REGION Network 2: Инициализация
   // При первом включении проверка наличия аварий и перегрева.
   // При перегреве --  охлаждение. Если долго не остывает, то авария.
   RUNG wire#powerrail
      "Initializing&Cooling_DB"(resetTrigg := wire#w1, iniOk => "Main_PRG".iniOk, initializing => "Main_PRG".initializing, faultTrigg => "READ".status.errorTrigg, warning => "READ".status.warning, toAirClean => #iniAir, toCoolUpLaser => #iniUpLaser, toCoolUpCam => #iniUpCam, toCoolDownLaser => #iniDownLaser, toCoolDownCam => #iniDownCam)
   END_RUNG
   RUNG wire#powerrail
      Contact( "WRITE".resetErrorTrigg )
   END_RUNG wire#w1
   RUNG wire#powerrail
      Contact( "READ".inputs.resetAlm )
   END_RUNG wire#w1
   // the same network as SCL:
   "Initializing&Cooling_DB"(resetTrigg := "WRITE".resetErrorTrigg OR "READ".inputs.resetAlm,   // "Initializing&Cooling"
                           iniOk => "Main_PRG".iniOk,
                           initializing => "Main_PRG".initializing,
                           faultTrigg => "READ".status.errorTrigg,
                           warning => "READ".status.warning,
                           toAirClean => #iniAir,
                           toCoolUpLaser => #iniUpLaser,
                           toCoolUpCam => #iniUpCam,
                           toCoolDownLaser => #iniDownLaser,
                           toCoolDownCam => #iniDownCam);
END_REGION

REGION Network 3: Основная программа
   // Включение велосиметра, обдува, охлаждения, сигналов ламп
   RUNG wire#powerrail
      "Main_Block_db"(faultTrigg := "READ".status.errorTrigg, warning := "READ".status.warning, initializing := "Main_PRG".initializing, initOk := "Main_PRG".iniOk, outEnable := "READ".inputs.runForward, velocimeterModeManual := "READ".inputs.veloModeManual, velocimeterModeAuto := "READ".inputs.veloModeAuto, revers := "READ".inputs.runBackward, synchroOn := "Main_PRG".synchroOn, airTon := "WRITE".cleanTime.tOnS, airToff := "WRITE".cleanTime.tOffMin, speed := "READ".velometer.instSpeed, RUN => "Main_PRG".RUN, airOn => #autoAir, veloLaser_En => "READ".outputs.disVelocimeter, veloShut_En => "READ".outputs.enVelocimeter, coolUpLaserOn => #autoUpLaser, coolUpCamOn => #autoUpCam, coolDownLaserOn => #autoDownLaser, coolDownCamOn => #autoDownCam, redLamp => "READ".outputs.redLamp, greenLamp => "READ".outputs.greenLamp, dirForward => "READ".status.veloPositive, dirBackward => "READ".status.veloNegative, greenLampStat => "READ".status.greenLamp, redLampStat => "READ".status.redLamp)
   END_RUNG
   // the same network as SCL:
   "Main_Block_db"(faultTrigg := "READ".status.errorTrigg,   // "Main_Block"
                   warning := "READ".status.warning,
                   initializing := "Main_PRG".initializing,
                   initOk := "Main_PRG".iniOk,
                   outEnable := "READ".inputs.runForward,
                   velocimeterModeManual := "READ".inputs.veloModeManual,
                   velocimeterModeAuto := "READ".inputs.veloModeAuto,
                   revers := "READ".inputs.runBackward,
                   synchroOn := "Main_PRG".synchroOn,
                   airTon := "WRITE".cleanTime.tOnS,
                   airToff := "WRITE".cleanTime.tOffMin,
                   speed := "READ".velometer.instSpeed,
                   RUN => "Main_PRG".RUN,
                   airOn => #autoAir,
                   veloLaser_En => "READ".outputs.disVelocimeter,
                   veloShut_En => "READ".outputs.enVelocimeter,
                   coolUpLaserOn => #autoUpLaser,
                   coolUpCamOn => #autoUpCam,
                   coolDownLaserOn => #autoDownLaser,
                   coolDownCamOn => #autoDownCam,
                   redLamp => "READ".outputs.redLamp,
                   greenLamp => "READ".outputs.greenLamp,
                   dirForward => "READ".status.veloPositive,
                   dirBackward => "READ".status.veloNegative,
                   greenLampStat => "READ".status.greenLamp,
                   redLampStat => "READ".status.redLamp);
END_REGION

REGION Network 4: Включение лазеров и синхронизации
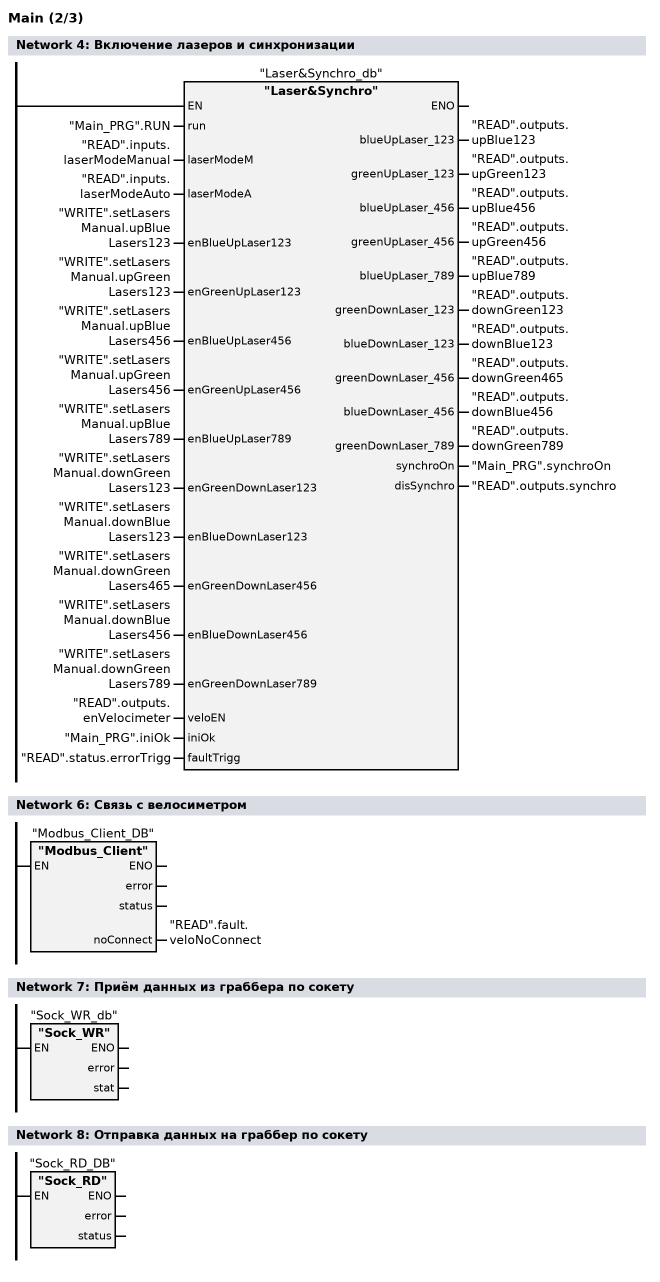
   RUNG wire#powerrail
      "Laser&Synchro_db"(run := "Main_PRG".RUN, laserModeM := "READ".inputs.laserModeManual, laserModeA := "READ".inputs.laserModeAuto, enBlueUpLaser123 := "WRITE".setLasersManual.upBlueLasers123, enGreenUpLaser123 := "WRITE".setLasersManual.upGreenLasers123, enBlueUpLaser456 := "WRITE".setLasersManual.upBlueLasers456, enGreenUpLaser456 := "WRITE".setLasersManual.upGreenLasers456, enBlueUpLaser789 := "WRITE".setLasersManual.upBlueLasers789, enGreenDownLaser123 := "WRITE".setLasersManual.downGreenLasers123, enBlueDownLaser123 := "WRITE".setLasersManual.downBlueLasers123, enGreenDownLaser456 := "WRITE".setLasersManual.downGreenLasers465, enBlueDownLaser456 := "WRITE".setLasersManual.downBlueLasers456, enGreenDownLaser789 := "WRITE".setLasersManual.downGreenLasers789, veloEN := "READ".outputs.enVelocimeter, iniOk := "Main_PRG".iniOk, faultTrigg := "READ".status.errorTrigg, blueUpLaser_123 => "READ".outputs.upBlue123, greenUpLaser_123 => "READ".outputs.upGreen123, blueUpLaser_456 => "READ".outputs.upBlue456, greenUpLaser_456 => "READ".outputs.upGreen456, blueUpLaser_789 => "READ".outputs.upBlue789, greenDownLaser_123 => "READ".outputs.downGreen123, blueDownLaser_123 => "READ".outputs.downBlue123, greenDownLaser_456 => "READ".outputs.downGreen465, blueDownLaser_456 => "READ".outputs.downBlue456, greenDownLaser_789 => "READ".outputs.downGreen789, synchroOn => "Main_PRG".synchroOn, disSynchro => "READ".outputs.synchro)
   END_RUNG
   // the same network as SCL:
   "Laser&Synchro_db"(run := "Main_PRG".RUN,   // "Laser&Synchro"
                      laserModeM := "READ".inputs.laserModeManual,
                      laserModeA := "READ".inputs.laserModeAuto,
                      enBlueUpLaser123 := "WRITE".setLasersManual.upBlueLasers123,
                      enGreenUpLaser123 := "WRITE".setLasersManual.upGreenLasers123,
                      enBlueUpLaser456 := "WRITE".setLasersManual.upBlueLasers456,
                      enGreenUpLaser456 := "WRITE".setLasersManual.upGreenLasers456,
                      enBlueUpLaser789 := "WRITE".setLasersManual.upBlueLasers789,
                      enGreenDownLaser123 := "WRITE".setLasersManual.downGreenLasers123,
                      enBlueDownLaser123 := "WRITE".setLasersManual.downBlueLasers123,
                      enGreenDownLaser456 := "WRITE".setLasersManual.downGreenLasers465,
                      enBlueDownLaser456 := "WRITE".setLasersManual.downBlueLasers456,
                      enGreenDownLaser789 := "WRITE".setLasersManual.downGreenLasers789,
                      veloEN := "READ".outputs.enVelocimeter,
                      iniOk := "Main_PRG".iniOk,
                      faultTrigg := "READ".status.errorTrigg,
                      blueUpLaser_123 => "READ".outputs.upBlue123,
                      greenUpLaser_123 => "READ".outputs.upGreen123,
                      blueUpLaser_456 => "READ".outputs.upBlue456,
                      greenUpLaser_456 => "READ".outputs.upGreen456,
                      blueUpLaser_789 => "READ".outputs.upBlue789,
                      greenDownLaser_123 => "READ".outputs.downGreen123,
                      blueDownLaser_123 => "READ".outputs.downBlue123,
                      greenDownLaser_456 => "READ".outputs.downGreen465,
                      blueDownLaser_456 => "READ".outputs.downBlue456,
                      greenDownLaser_789 => "READ".outputs.downGreen789,
                      synchroOn => "Main_PRG".synchroOn,
                      disSynchro => "READ".outputs.synchro);
END_REGION

REGION Network 5 (SCL): Объединение сигналов
   "READ".outputs.airClean := #iniAir OR #autoAir;
   "READ".outputs.coolUpLaser := #iniUpLaser OR #autoUpLaser;
   "READ".outputs.coolUpCam := #iniUpCam OR #autoUpCam;
   "READ".outputs.coolDownLaser := #iniDownLaser OR #autoDownLaser;
   "READ".outputs.coolDownCam := #iniDownCam OR #autoDownCam;
END_REGION

REGION Network 6: Связь с велосиметром
   RUNG wire#powerrail
      "Modbus_Client_DB"(error =>, status =>, noConnect => "READ".fault.veloNoConnect)
   END_RUNG
   // the same network as SCL:
   "Modbus_Client_DB"(noConnect => "READ".fault.veloNoConnect);   // "Modbus_Client"
END_REGION

REGION Network 7: Приём данных из граббера по сокету
   RUNG wire#powerrail
      "Sock_WR_db"(error =>, stat =>)
   END_RUNG
   // the same network as SCL:
   "Sock_WR_db"();   // "Sock_WR"
END_REGION

REGION Network 8: Отправка данных на граббер по сокету
   RUNG wire#powerrail
      "Sock_RD_DB"(error =>, status =>)
   END_RUNG
   // the same network as SCL:
   "Sock_RD_DB"();   // "Sock_RD"
END_REGION

REGION Network 9: Включение охладителя воздуха пневмосистемы
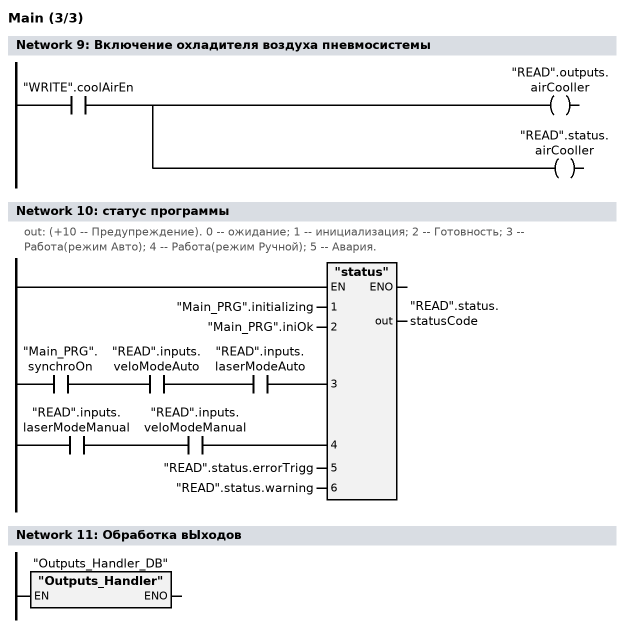
   RUNG wire#powerrail
      Contact( "WRITE".coolAirEn )
      wire#w1
      Coil( "READ".outputs.airCooller )
   END_RUNG
   RUNG wire#w1
      Coil( "READ".status.airCooller )
   END_RUNG
   // the same network as SCL:
   "READ".outputs.airCooller := "WRITE".coolAirEn;
   "READ".status.airCooller := "WRITE".coolAirEn;
END_REGION

REGION Network 10: статус программы
   // out: (+10 -- Предупреждение). 0 -- ожидание; 1 -- инициализация; 2 -- Готовность; 3 -- Работа(режим Авто); 4 -- Работа(режим Ручной); 5 -- Авария.
   RUNG wire#powerrail
      "status"("3" := wire#w1, "4" := wire#w2, "1" := "Main_PRG".initializing, "2" := "Main_PRG".iniOk, "5" := "READ".status.errorTrigg, "6" := "READ".status.warning, out => "READ".status.statusCode)
   END_RUNG
   RUNG wire#powerrail
      Contact( "Main_PRG".synchroOn )
      Contact( "READ".inputs.veloModeAuto )
      Contact( "READ".inputs.laserModeAuto )
   END_RUNG wire#w1
   RUNG wire#powerrail
      Contact( "READ".inputs.laserModeManual )
      Contact( "READ".inputs.veloModeManual )
   END_RUNG wire#w2
   // the same network as SCL:
   "status"("1" := "Main_PRG".initializing,
            "2" := "Main_PRG".iniOk,
            "3" := "Main_PRG".synchroOn AND "READ".inputs.veloModeAuto AND "READ".inputs.laserModeAuto,
            "4" := "READ".inputs.laserModeManual AND "READ".inputs.veloModeManual,
            "5" := "READ".status.errorTrigg,
            "6" := "READ".status.warning,
            out => "READ".status.statusCode);
END_REGION

REGION Network 11: Обработка вЫходов
   RUNG wire#powerrail
      "Outputs_Handler_DB"()
   END_RUNG
   // the same network as SCL:
   "Outputs_Handler_DB"();   // "Outputs_Handler"
END_REGION
END_ORGANIZATION_BLOCK

// folder: FBlocks

FUNCTION_BLOCK "Decode8toBool"   // FB2, SCL
{ S7_Optimized_Access := 'TRUE' }
VERSION : 0.1
   VAR_INPUT
      in : Byte;
   END_VAR
   VAR_OUTPUT
      b0 : Bool;
      b1 : Bool;
      b2 : Bool;
      b3 : Bool;
      b4 : Bool;
      b5 : Bool;
      b6 : Bool;
      b7 : Bool;
      "OR" : Bool;
   END_VAR
   VAR
      boolArray : Array[0..7] of Bool;
      i : USInt;
      "m" : USInt;
      temp : UDInt;
   END_VAR
BEGIN
   FOR #i := 0 TO 7 DO
       "MOD"(in0 := #in,
             in1 := 2,
             Out => #m);
       IF #m > 0 THEN
           #boolArray[#i] := TRUE;
       ELSE
           #boolArray[#i] := FALSE;
       END_IF;
       #in := #in / 2;
   END_FOR;

   #b0 := #boolArray[0];
   #b1 := #boolArray[1];
   #b2 := #boolArray[2];
   #b3 := #boolArray[3];
   #b4 := #boolArray[4];
   #b5 := #boolArray[5];
   #b6 := #boolArray[6];
   #b7 := #boolArray[7];

   #OR := #b2 OR #b4 OR #b6 OR #b7;
END_FUNCTION_BLOCK

FUNCTION_BLOCK "Hysteresis"   // FB4, LAD
{ S7_Optimized_Access := 'TRUE' }
VERSION : 0.1
   VAR_INPUT
      in : Real;
      SP : Real;
      hyster : Real;
   END_VAR
   VAR_OUTPUT
      cold : Bool;
      warm : Bool;
   END_VAR
   VAR_TEMP
      upperThreshold : Real;
      lowerThreshold : Real;
   END_VAR
BEGIN

REGION Network 1 (SCL)
   #upperThreshold := #SP + (#hyster / 2);
   #lowerThreshold := #SP - (#hyster / 2);

   IF #in > #upperThreshold THEN
       #cold := true;
       #warm := false;
   ELSIF #in < #lowerThreshold THEN
       #cold := false;
       #warm := true;
   END_IF;
END_REGION
END_FUNCTION_BLOCK

FUNCTION_BLOCK "4Hysteresis"   // FB5, LAD
{ S7_Optimized_Access := 'TRUE' }
VERSION : 0.1
   VAR_INPUT
      in0 : Real;
      in1 : Real := 0.0;
      in2 : Real := 0.0;
      in3 : Real := 0.0;
      SP0 : Real;
      SP1 : Real := 0.0;
      SP2 : Real := 0.0;
      SP3 : Real := 0.0;
      hyster : Real;
      TON : Time;
   END_VAR
   VAR_OUTPUT
      out0 : Bool;
      out1 : Bool := false;
      out2 : Bool := false;
      out3 : Bool := false;
   END_VAR
   VAR
      Hysteresis_Instance : "Hysteresis";
      Hysteresis_Instance_1 : "Hysteresis";
      Hysteresis_Instance_2 : "Hysteresis";
      Hysteresis_Instance_3 : "Hysteresis";
      IEC_Timer_0_Instance : TON_TIME;
      IEC_Timer_0_Instance_1 : TON_TIME;
      IEC_Timer_0_Instance_2 : TON_TIME;
      IEC_Timer_0_Instance_3 : TON_TIME;
   END_VAR
   VAR_TEMP
      gi0 : Bool;
      gi1 : Bool;
      gi2 : Bool;
      gi3 : Bool;
   END_VAR
BEGIN

REGION Network 1
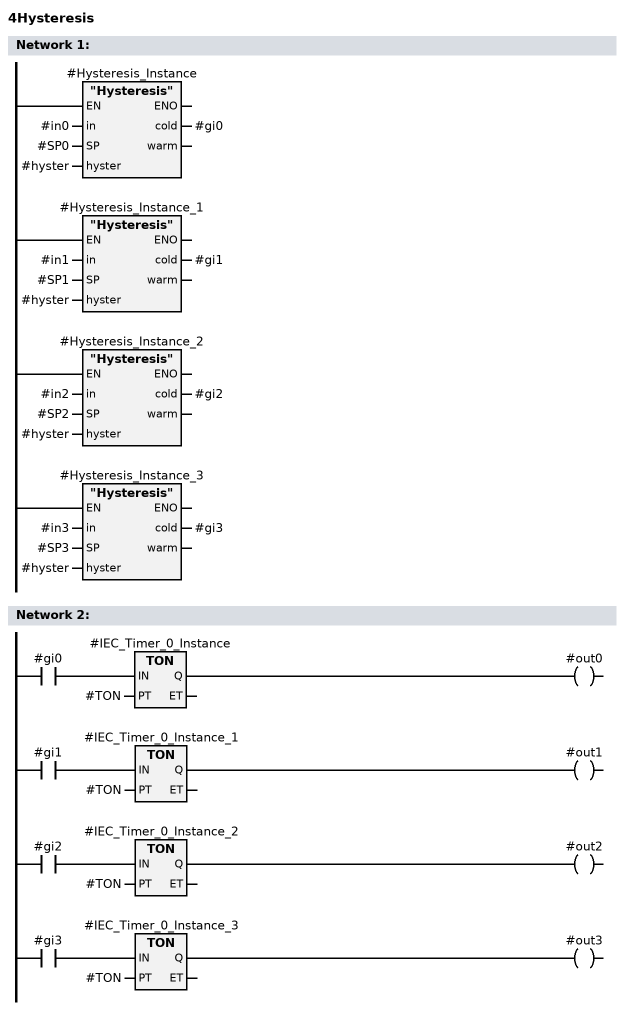
   RUNG wire#powerrail
      #Hysteresis_Instance(in := #in0, SP := #SP0, hyster := #hyster, cold => #gi0, warm =>)
   END_RUNG
   RUNG wire#powerrail
      #Hysteresis_Instance_1(in := #in1, SP := #SP1, hyster := #hyster, cold => #gi1, warm =>)
   END_RUNG
   RUNG wire#powerrail
      #Hysteresis_Instance_2(in := #in2, SP := #SP2, hyster := #hyster, cold => #gi2, warm =>)
   END_RUNG
   RUNG wire#powerrail
      #Hysteresis_Instance_3(in := #in3, SP := #SP3, hyster := #hyster, cold => #gi3, warm =>)
   END_RUNG
   // the same network as SCL:
   #Hysteresis_Instance(in := #in0, SP := #SP0, hyster := #hyster, cold => #gi0);   // "Hysteresis"
   #Hysteresis_Instance_1(in := #in1, SP := #SP1, hyster := #hyster, cold => #gi1);   // "Hysteresis"
   #Hysteresis_Instance_2(in := #in2, SP := #SP2, hyster := #hyster, cold => #gi2);   // "Hysteresis"
   #Hysteresis_Instance_3(in := #in3, SP := #SP3, hyster := #hyster, cold => #gi3);   // "Hysteresis"
END_REGION

REGION Network 2
   #IEC_Timer_0_Instance(IN := #gi0, PT := #TON);   // TON
   #out0 := #IEC_Timer_0_Instance.Q;
   #IEC_Timer_0_Instance_1(IN := #gi1, PT := #TON);   // TON
   #out1 := #IEC_Timer_0_Instance_1.Q;
   #IEC_Timer_0_Instance_2(IN := #gi2, PT := #TON);   // TON
   #out2 := #IEC_Timer_0_Instance_2.Q;
   #IEC_Timer_0_Instance_3(IN := #gi3, PT := #TON);   // TON
   #out3 := #IEC_Timer_0_Instance_3.Q;
END_REGION
END_FUNCTION_BLOCK

FUNCTION_BLOCK "5Hysteresis"   // FB6, LAD
{ S7_Optimized_Access := 'TRUE' }
VERSION : 0.1
   VAR_INPUT
      in0 : Real;
      in1 : Real := 0.0;
      in2 : Real := 0.0;
      in3 : Real := 0.0;
      in4 : Real := 0.0;
      SP0 : Real;
      SP1 : Real := 0.0;
      SP2 : Real := 0.0;
      SP3 : Real := 0.0;
      SP4 : Real := 0.0;
      hyster : Real;
   END_VAR
   VAR_OUTPUT
      out0 : Bool;
      out1 : Bool := false;
      out2 : Bool := false;
      out3 : Bool := false;
      out4 : Bool := false;
   END_VAR
   VAR
      Hysteresis_Instance : "Hysteresis";
      Hysteresis_Instance_1 : "Hysteresis";
      Hysteresis_Instance_2 : "Hysteresis";
      Hysteresis_Instance_3 : "Hysteresis";
      Hysteresis_Instance_4 : "Hysteresis";
   END_VAR
BEGIN

REGION Network 1
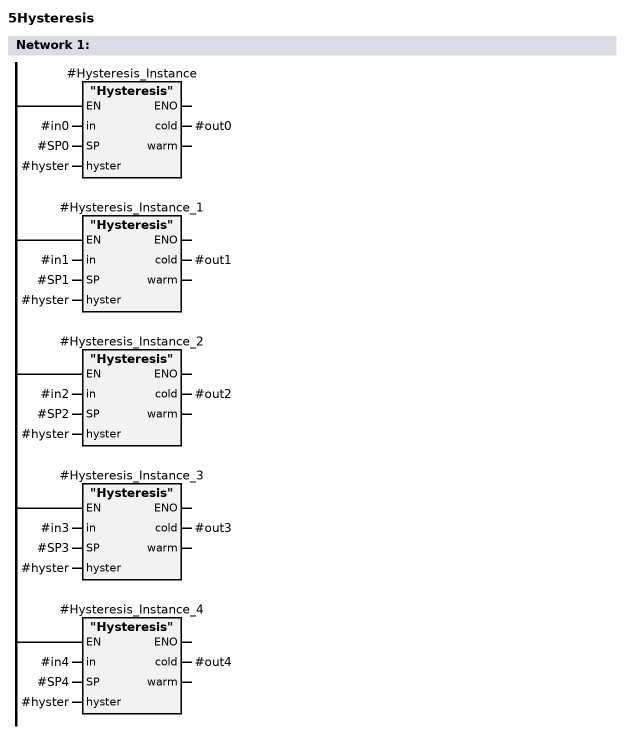
   RUNG wire#powerrail
      #Hysteresis_Instance(in := #in0, SP := #SP0, hyster := #hyster, cold => #out0, warm =>)
   END_RUNG
   RUNG wire#powerrail
      #Hysteresis_Instance_1(in := #in1, SP := #SP1, hyster := #hyster, cold => #out1, warm =>)
   END_RUNG
   RUNG wire#powerrail
      #Hysteresis_Instance_2(in := #in2, SP := #SP2, hyster := #hyster, cold => #out2, warm =>)
   END_RUNG
   RUNG wire#powerrail
      #Hysteresis_Instance_3(in := #in3, SP := #SP3, hyster := #hyster, cold => #out3, warm =>)
   END_RUNG
   RUNG wire#powerrail
      #Hysteresis_Instance_4(in := #in4, SP := #SP4, hyster := #hyster, cold => #out4, warm =>)
   END_RUNG
   // the same network as SCL:
   #Hysteresis_Instance(in := #in0, SP := #SP0, hyster := #hyster, cold => #out0);   // "Hysteresis"
   #Hysteresis_Instance_1(in := #in1, SP := #SP1, hyster := #hyster, cold => #out1);   // "Hysteresis"
   #Hysteresis_Instance_2(in := #in2, SP := #SP2, hyster := #hyster, cold => #out2);   // "Hysteresis"
   #Hysteresis_Instance_3(in := #in3, SP := #SP3, hyster := #hyster, cold => #out3);   // "Hysteresis"
   #Hysteresis_Instance_4(in := #in4, SP := #SP4, hyster := #hyster, cold => #out4);   // "Hysteresis"
END_REGION
END_FUNCTION_BLOCK

FUNCTION_BLOCK "initializing"   // FB8, LAD
{ S7_Optimized_Access := 'TRUE' }
VERSION : 0.1
   VAR_INPUT
      warnTempUpLaser : Bool;
      warnTempUpCam : Bool;
      warnTempDowLaser : Bool;
      warnTempDowCam : Bool;
      reset : Bool;
      coolErrTime : Time;
   END_VAR
   VAR_OUTPUT
      iniOk : Bool;
      Initia : Bool;
      iniErr : Bool;
      airClean : Bool;
      toCoolUpLaser : Bool;
      toCoolUpCam : Bool;
      toCoolDownLaser : Bool;
      toCoolDownCam : Bool;
   END_VAR
   VAR
      IEC_Timer_0_Instance : TON_TIME;
      cleaned : Bool;
      rise0 : Bool;
      fall0 : Bool;
      t0 : Bool;
      IEC_Timer_0_Instance_1 : TON_TIME;
      IEC_Timer_0_Instance_2 : TOF_TIME;
      IEC_Timer_0_Instance_3 : TOF_TIME;
   END_VAR
   VAR_TEMP
      firstStart : Bool;
      tempOk : Bool;
      coolErr : Bool;
      TOF_firstStart : Bool;
      temperaturesOK : Bool;
   END_VAR
   VAR_TEMP   // added for the SCL form of the ladder/FBD networks
      _w1 : Bool;
      _w2 : Bool;
   END_VAR
BEGIN

REGION Network 1: Первая очистка
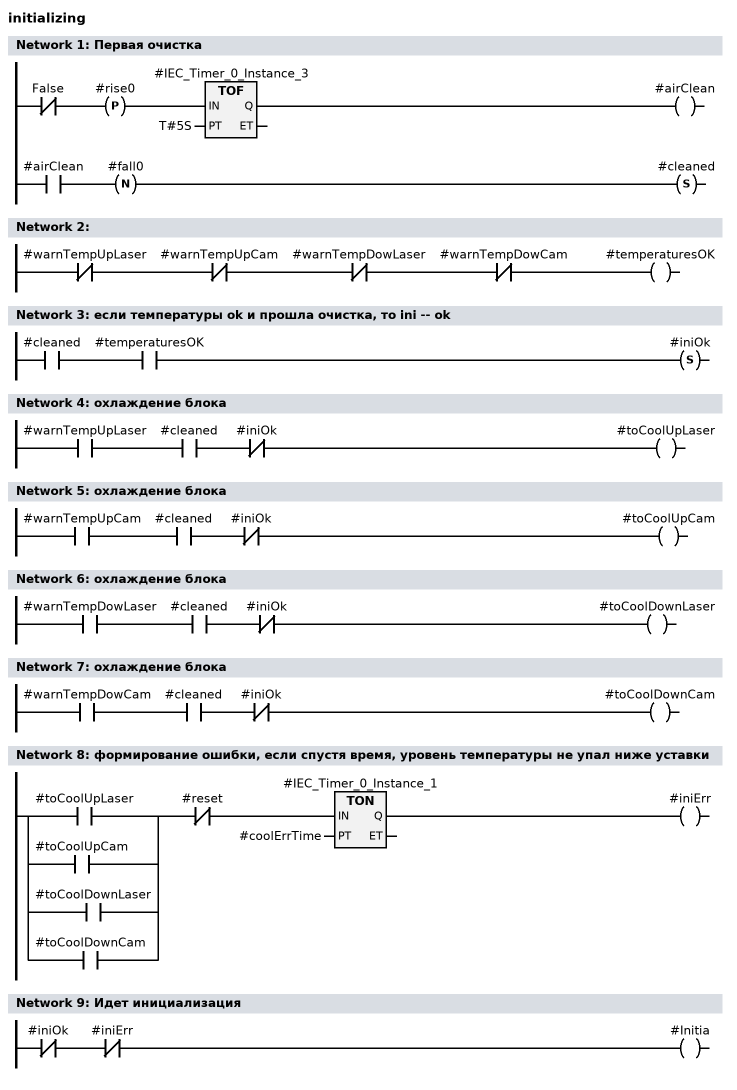
   #_w1 := NOT False AND NOT #rise0;   // rising edge
   #rise0 := NOT False;
   #IEC_Timer_0_Instance_3(IN := #_w1, PT := T#5S);   // TOF
   #airClean := #IEC_Timer_0_Instance_3.Q;
   #_w2 := NOT #airClean AND #fall0;   // falling edge
   #fall0 := #airClean;
   IF #_w2 THEN #cleaned := TRUE; END_IF;
END_REGION

REGION Network 2
   RUNG wire#powerrail
      I_Contact( #warnTempUpLaser )
      I_Contact( #warnTempUpCam )
      I_Contact( #warnTempDowLaser )
      I_Contact( #warnTempDowCam )
      Coil( #temperaturesOK )
   END_RUNG
   // the same network as SCL:
   #temperaturesOK := NOT #warnTempUpLaser AND NOT #warnTempUpCam AND NOT #warnTempDowLaser AND NOT #warnTempDowCam;
END_REGION

REGION Network 3: если температуры ok и прошла очистка, то ini -- ok
   RUNG wire#powerrail
      Contact( #cleaned )
      Contact( #temperaturesOK )
      S_Coil( #iniOk )
   END_RUNG
   // the same network as SCL:
   IF #cleaned AND #temperaturesOK THEN #iniOk := TRUE; END_IF;
END_REGION

REGION Network 4: охлаждение блока
   RUNG wire#powerrail
      Contact( #warnTempUpLaser )
      Contact( #cleaned )
      I_Contact( #iniOk )
      Coil( #toCoolUpLaser )
   END_RUNG
   // the same network as SCL:
   #toCoolUpLaser := #warnTempUpLaser AND #cleaned AND NOT #iniOk;
END_REGION

REGION Network 5: охлаждение блока
   RUNG wire#powerrail
      Contact( #warnTempUpCam )
      Contact( #cleaned )
      I_Contact( #iniOk )
      Coil( #toCoolUpCam )
   END_RUNG
   // the same network as SCL:
   #toCoolUpCam := #warnTempUpCam AND #cleaned AND NOT #iniOk;
END_REGION

REGION Network 6: охлаждение блока
   RUNG wire#powerrail
      Contact( #warnTempDowLaser )
      Contact( #cleaned )
      I_Contact( #iniOk )
      Coil( #toCoolDownLaser )
   END_RUNG
   // the same network as SCL:
   #toCoolDownLaser := #warnTempDowLaser AND #cleaned AND NOT #iniOk;
END_REGION

REGION Network 7: охлаждение блока
   RUNG wire#powerrail
      Contact( #warnTempDowCam )
      Contact( #cleaned )
      I_Contact( #iniOk )
      Coil( #toCoolDownCam )
   END_RUNG
   // the same network as SCL:
   #toCoolDownCam := #warnTempDowCam AND #cleaned AND NOT #iniOk;
END_REGION

REGION Network 8: формирование ошибки, если спустя время, уровень температуры не упал ниже уставки
   #IEC_Timer_0_Instance_1(IN := (#toCoolUpLaser OR #toCoolUpCam OR #toCoolDownLaser OR #toCoolDownCam) AND NOT #reset,   // TON
                           PT := #coolErrTime);
   #iniErr := #IEC_Timer_0_Instance_1.Q;
END_REGION

REGION Network 9: Идет инициализация
   RUNG wire#powerrail
      I_Contact( #iniOk )
      I_Contact( #iniErr )
      Coil( #Initia )
   END_RUNG
   // the same network as SCL:
   #Initia := NOT #iniOk AND NOT #iniErr;
END_REGION
END_FUNCTION_BLOCK

FUNCTION_BLOCK "Blink"   // FB10, LAD
{ S7_Optimized_Access := 'TRUE' }
VERSION : 0.1
   VAR_INPUT
      in : Bool;
      Ton : DInt;
      Toff : DInt;
   END_VAR
   VAR_OUTPUT
      Q : Bool;
   END_VAR
   VAR
      t0 : Bool;
      IEC_Timer_0_Instance : TON_TIME;
      IEC_Timer_0_Instance_1 : TON_TIME;
   END_VAR
   VAR_TEMP
      t1 : Bool;
   END_VAR
   VAR_TEMP   // added for the SCL form of the ladder/FBD networks
      _w1 : Bool;
   END_VAR
BEGIN

REGION Network 1
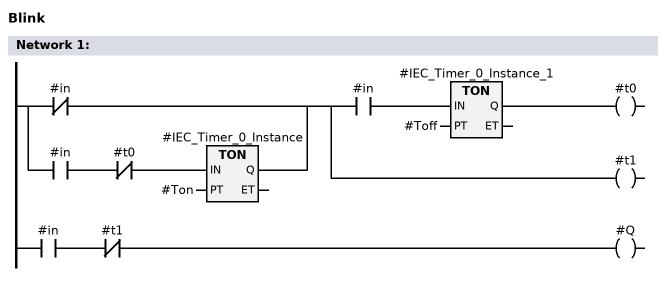
   #IEC_Timer_0_Instance(IN := #in AND NOT #t0, PT := #Ton);   // TON
   #_w1 := NOT #in OR #IEC_Timer_0_Instance.Q;
   #IEC_Timer_0_Instance_1(IN := #_w1 AND #in, PT := #Toff);   // TON
   #t0 := #IEC_Timer_0_Instance_1.Q;
   #t1 := #_w1;
   #Q := #in AND NOT #t1;
END_REGION
END_FUNCTION_BLOCK

FUNCTION_BLOCK "ChangeReal"   // FB14, SCL
{ S7_Optimized_Access := 'TRUE' }
VERSION : 0.1
   VAR_INPUT
      in : Real;
   END_VAR
   VAR_OUTPUT
      "^out" : Bool;
   END_VAR
   VAR
      buff : Real;
   END_VAR
BEGIN
   IF #in <> #buff THEN
       #"^out" := true;
   ELSE
       #"^out" := false;
   END_IF;
   #buff := #in;
END_FUNCTION_BLOCK

// folder: Functions

FUNCTION "DI_simulate" : Void   // FC1, LAD
{ S7_Optimized_Access := 'TRUE' }
VERSION : 0.1
   VAR_INPUT
      in0 : Bool;
      in1 : Bool;
      in2 : Bool;
      in3 : Bool;
      in4 : Bool;
      in5 : Bool;
      in6 : Bool;
      in7 : Bool;
      in8 : Bool;
      in9 : Bool;
      in10 : Bool;
      in11 : Bool;
      in12 : Bool;
      in13 : Bool;
      in14 : Bool;
      in15 : Bool;
      inSimulate : Struct
         DI0 : USInt;
         DI1 : USInt;
         DI2 : USInt;
         DI3 : USInt;
         DI4 : USInt;
         DI5 : USInt;
         DI6 : USInt;
         DI7 : USInt;
         DI8 : USInt;
         DI9 : USInt;
         DI10 : USInt;
         DI11 : USInt;
         DI12 : USInt;
         DI13 : USInt;
         DI14 : USInt;
         DI15 : USInt;
      END_STRUCT;
   END_VAR
   VAR_OUTPUT
      out0 : Bool;
      out1 : Bool;
      out2 : Bool;
      out3 : Bool;
      out4 : Bool;
      out5 : Bool;
      out6 : Bool;
      out7 : Bool;
      out8 : Bool;
      out9 : Bool;
      out10 : Bool;
      out11 : Bool;
      out12 : Bool;
      out13 : Bool;
      out14 : Bool;
      out15 : Bool;
   END_VAR
BEGIN

REGION Network 1
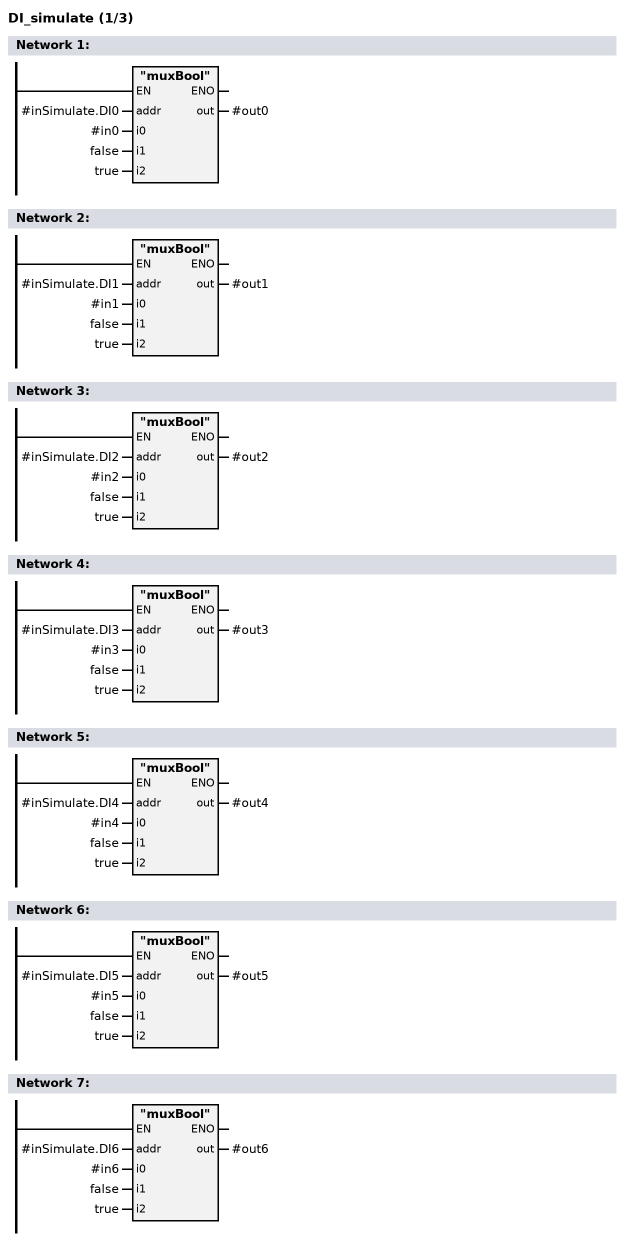
   RUNG wire#powerrail
      "muxBool"(addr := #inSimulate.DI0, i0 := #in0, i1 := false, i2 := true, out => #out0)
   END_RUNG
   // the same network as SCL:
   "muxBool"(addr := #inSimulate.DI0, i0 := #in0, i1 := false, i2 := true, out => #out0);
END_REGION

REGION Network 2
   RUNG wire#powerrail
      "muxBool"(addr := #inSimulate.DI1, i0 := #in1, i1 := false, i2 := true, out => #out1)
   END_RUNG
   // the same network as SCL:
   "muxBool"(addr := #inSimulate.DI1, i0 := #in1, i1 := false, i2 := true, out => #out1);
END_REGION

REGION Network 3
   RUNG wire#powerrail
      "muxBool"(addr := #inSimulate.DI2, i0 := #in2, i1 := false, i2 := true, out => #out2)
   END_RUNG
   // the same network as SCL:
   "muxBool"(addr := #inSimulate.DI2, i0 := #in2, i1 := false, i2 := true, out => #out2);
END_REGION

REGION Network 4
   RUNG wire#powerrail
      "muxBool"(addr := #inSimulate.DI3, i0 := #in3, i1 := false, i2 := true, out => #out3)
   END_RUNG
   // the same network as SCL:
   "muxBool"(addr := #inSimulate.DI3, i0 := #in3, i1 := false, i2 := true, out => #out3);
END_REGION

REGION Network 5
   RUNG wire#powerrail
      "muxBool"(addr := #inSimulate.DI4, i0 := #in4, i1 := false, i2 := true, out => #out4)
   END_RUNG
   // the same network as SCL:
   "muxBool"(addr := #inSimulate.DI4, i0 := #in4, i1 := false, i2 := true, out => #out4);
END_REGION

REGION Network 6
   RUNG wire#powerrail
      "muxBool"(addr := #inSimulate.DI5, i0 := #in5, i1 := false, i2 := true, out => #out5)
   END_RUNG
   // the same network as SCL:
   "muxBool"(addr := #inSimulate.DI5, i0 := #in5, i1 := false, i2 := true, out => #out5);
END_REGION

REGION Network 7
   RUNG wire#powerrail
      "muxBool"(addr := #inSimulate.DI6, i0 := #in6, i1 := false, i2 := true, out => #out6)
   END_RUNG
   // the same network as SCL:
   "muxBool"(addr := #inSimulate.DI6, i0 := #in6, i1 := false, i2 := true, out => #out6);
END_REGION

REGION Network 8
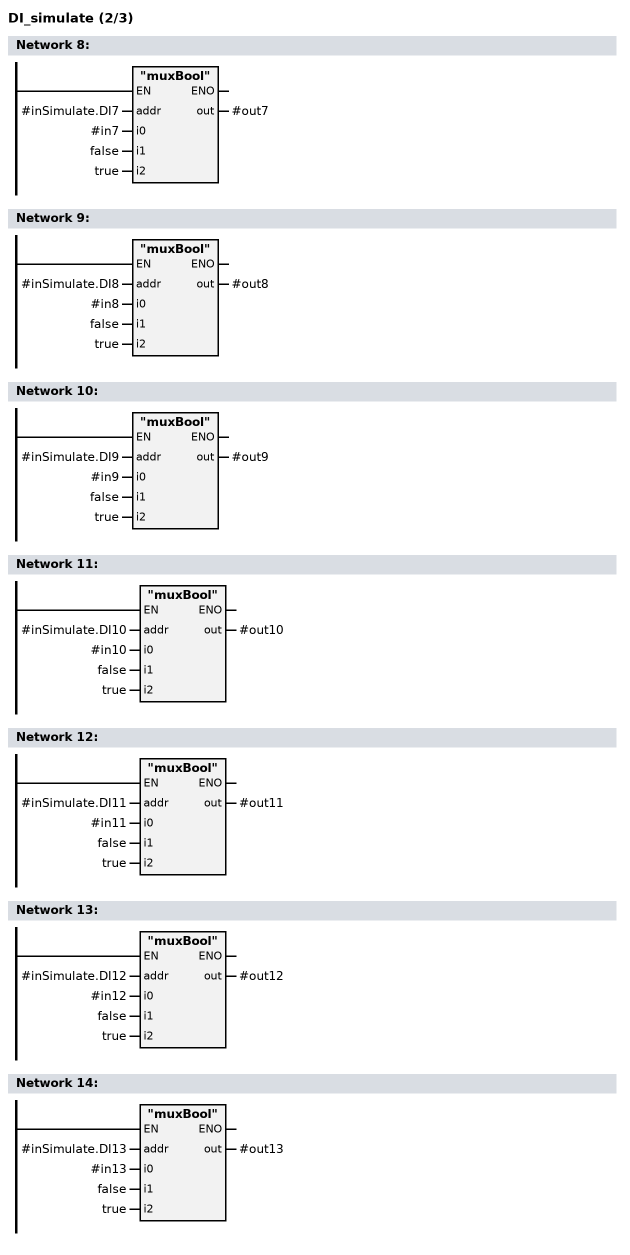
   RUNG wire#powerrail
      "muxBool"(addr := #inSimulate.DI7, i0 := #in7, i1 := false, i2 := true, out => #out7)
   END_RUNG
   // the same network as SCL:
   "muxBool"(addr := #inSimulate.DI7, i0 := #in7, i1 := false, i2 := true, out => #out7);
END_REGION

REGION Network 9
   RUNG wire#powerrail
      "muxBool"(addr := #inSimulate.DI8, i0 := #in8, i1 := false, i2 := true, out => #out8)
   END_RUNG
   // the same network as SCL:
   "muxBool"(addr := #inSimulate.DI8, i0 := #in8, i1 := false, i2 := true, out => #out8);
END_REGION

REGION Network 10
   RUNG wire#powerrail
      "muxBool"(addr := #inSimulate.DI9, i0 := #in9, i1 := false, i2 := true, out => #out9)
   END_RUNG
   // the same network as SCL:
   "muxBool"(addr := #inSimulate.DI9, i0 := #in9, i1 := false, i2 := true, out => #out9);
END_REGION

REGION Network 11
   RUNG wire#powerrail
      "muxBool"(addr := #inSimulate.DI10, i0 := #in10, i1 := false, i2 := true, out => #out10)
   END_RUNG
   // the same network as SCL:
   "muxBool"(addr := #inSimulate.DI10, i0 := #in10, i1 := false, i2 := true, out => #out10);
END_REGION

REGION Network 12
   RUNG wire#powerrail
      "muxBool"(addr := #inSimulate.DI11, i0 := #in11, i1 := false, i2 := true, out => #out11)
   END_RUNG
   // the same network as SCL:
   "muxBool"(addr := #inSimulate.DI11, i0 := #in11, i1 := false, i2 := true, out => #out11);
END_REGION

REGION Network 13
   RUNG wire#powerrail
      "muxBool"(addr := #inSimulate.DI12, i0 := #in12, i1 := false, i2 := true, out => #out12)
   END_RUNG
   // the same network as SCL:
   "muxBool"(addr := #inSimulate.DI12, i0 := #in12, i1 := false, i2 := true, out => #out12);
END_REGION

REGION Network 14
   RUNG wire#powerrail
      "muxBool"(addr := #inSimulate.DI13, i0 := #in13, i1 := false, i2 := true, out => #out13)
   END_RUNG
   // the same network as SCL:
   "muxBool"(addr := #inSimulate.DI13, i0 := #in13, i1 := false, i2 := true, out => #out13);
END_REGION

REGION Network 15
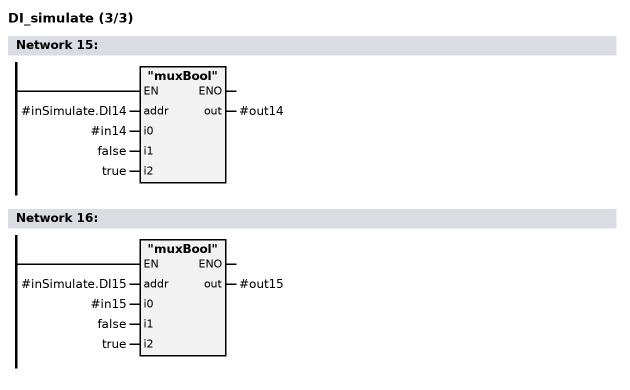
   RUNG wire#powerrail
      "muxBool"(addr := #inSimulate.DI14, i0 := #in14, i1 := false, i2 := true, out => #out14)
   END_RUNG
   // the same network as SCL:
   "muxBool"(addr := #inSimulate.DI14, i0 := #in14, i1 := false, i2 := true, out => #out14);
END_REGION

REGION Network 16
   RUNG wire#powerrail
      "muxBool"(addr := #inSimulate.DI15, i0 := #in15, i1 := false, i2 := true, out => #out15)
   END_RUNG
   // the same network as SCL:
   "muxBool"(addr := #inSimulate.DI15, i0 := #in15, i1 := false, i2 := true, out => #out15);
END_REGION
END_FUNCTION

FUNCTION "DO_simulate" : Void   // FC2, LAD
{ S7_Optimized_Access := 'TRUE' }
VERSION : 0.1
   VAR_INPUT
      in0 : Bool;
      in1 : Bool;
      in2 : Bool;
      in3 : Bool;
      in4 : Bool;
      in5 : Bool;
      in6 : Bool;
      in7 : Bool;
      in8 : Bool;
      in9 : Bool;
      in10 : Bool;
      in11 : Bool;
      in12 : Bool;
      in13 : Bool;
      in14 : Bool;
      in15 : Bool;
      in16 : Bool;
      in17 : Bool;
      in18 : Bool;
      in19 : Bool;
      in20 : Bool;
      in21 : Bool;
      inSimulate : Struct
         DO0 : USInt;
         DO1 : USInt;
         DO2 : USInt;
         DO3 : USInt;
         DO4 : USInt;
         DO5 : USInt;
         DO6 : USInt;
         DO7 : USInt;
         DO8 : USInt;
         DO9 : USInt;
         DO10 : USInt;
         DO11 : USInt;
         DO12 : USInt;
         DO13 : USInt;
         DO14 : USInt;
         DO15 : USInt;
         DO16 : USInt;
         DO17 : USInt;
         DO18 : USInt;
         DO19 : USInt;
         DO20 : USInt;
         DO21 : USInt;
         DO22 : USInt;
         DO23 : USInt;
         DO24 : USInt;
         DO25 : USInt;
         DO26 : USInt;
         DO27 : USInt;
         DO28 : USInt;
         DO29 : USInt;
         DO30 : USInt;
         DO31 : USInt;
      END_STRUCT;
   END_VAR
   VAR_OUTPUT
      out0 : Bool;
      out1 : Bool;
      out2 : Bool;
      out3 : Bool;
      out4 : Bool;
      out5 : Bool;
      out6 : Bool;
      out7 : Bool;
      out8 : Bool;
      out9 : Bool;
      out10 : Bool;
      out11 : Bool;
      out12 : Bool;
      out13 : Bool;
      out14 : Bool;
      out15 : Bool;
      out16 : Bool;
      out17 : Bool;
      out18 : Bool;
      out19 : Bool;
      out20 : Bool;
      out21 : Bool;
   END_VAR
BEGIN

REGION Network 2
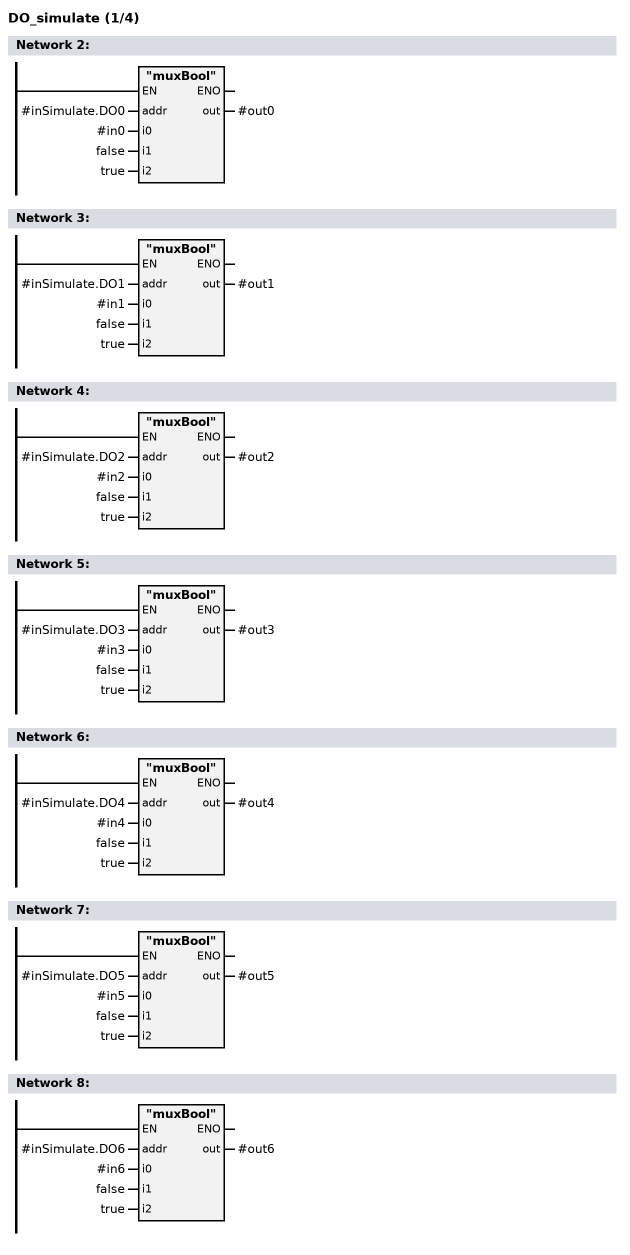
   RUNG wire#powerrail
      "muxBool"(addr := #inSimulate.DO0, i0 := #in0, i1 := false, i2 := true, out => #out0)
   END_RUNG
   // the same network as SCL:
   "muxBool"(addr := #inSimulate.DO0, i0 := #in0, i1 := false, i2 := true, out => #out0);
END_REGION

REGION Network 3
   RUNG wire#powerrail
      "muxBool"(addr := #inSimulate.DO1, i0 := #in1, i1 := false, i2 := true, out => #out1)
   END_RUNG
   // the same network as SCL:
   "muxBool"(addr := #inSimulate.DO1, i0 := #in1, i1 := false, i2 := true, out => #out1);
END_REGION

REGION Network 4
   RUNG wire#powerrail
      "muxBool"(addr := #inSimulate.DO2, i0 := #in2, i1 := false, i2 := true, out => #out2)
   END_RUNG
   // the same network as SCL:
   "muxBool"(addr := #inSimulate.DO2, i0 := #in2, i1 := false, i2 := true, out => #out2);
END_REGION

REGION Network 5
   RUNG wire#powerrail
      "muxBool"(addr := #inSimulate.DO3, i0 := #in3, i1 := false, i2 := true, out => #out3)
   END_RUNG
   // the same network as SCL:
   "muxBool"(addr := #inSimulate.DO3, i0 := #in3, i1 := false, i2 := true, out => #out3);
END_REGION

REGION Network 6
   RUNG wire#powerrail
      "muxBool"(addr := #inSimulate.DO4, i0 := #in4, i1 := false, i2 := true, out => #out4)
   END_RUNG
   // the same network as SCL:
   "muxBool"(addr := #inSimulate.DO4, i0 := #in4, i1 := false, i2 := true, out => #out4);
END_REGION

REGION Network 7
   RUNG wire#powerrail
      "muxBool"(addr := #inSimulate.DO5, i0 := #in5, i1 := false, i2 := true, out => #out5)
   END_RUNG
   // the same network as SCL:
   "muxBool"(addr := #inSimulate.DO5, i0 := #in5, i1 := false, i2 := true, out => #out5);
END_REGION

REGION Network 8
   RUNG wire#powerrail
      "muxBool"(addr := #inSimulate.DO6, i0 := #in6, i1 := false, i2 := true, out => #out6)
   END_RUNG
   // the same network as SCL:
   "muxBool"(addr := #inSimulate.DO6, i0 := #in6, i1 := false, i2 := true, out => #out6);
END_REGION

REGION Network 9
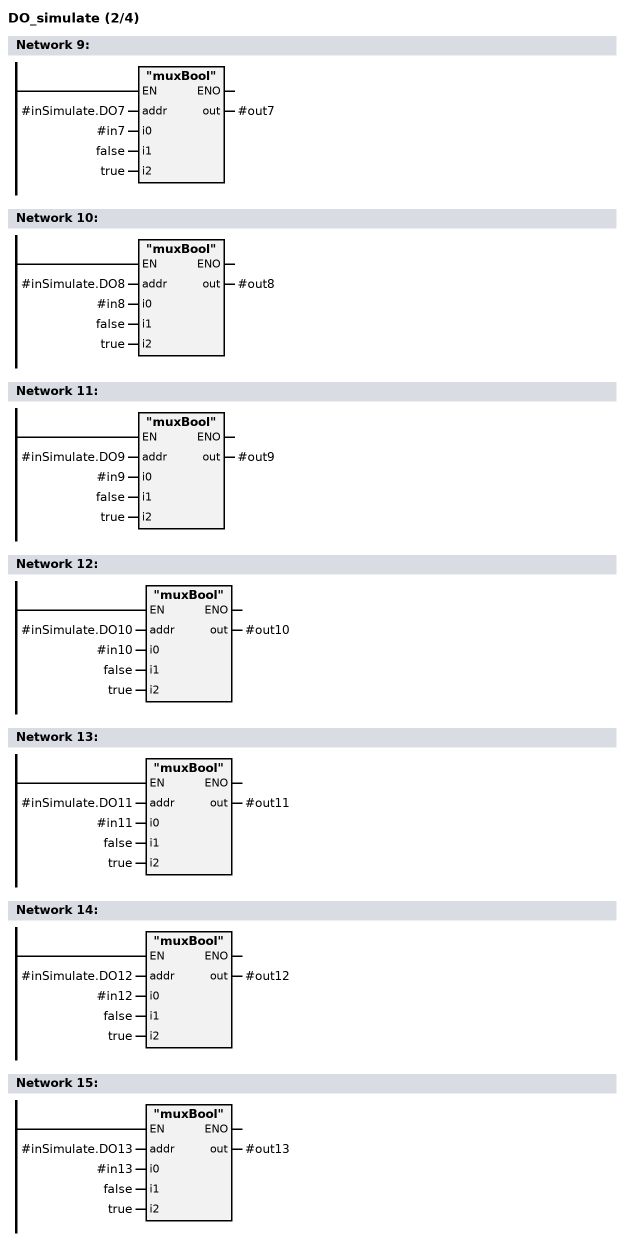
   RUNG wire#powerrail
      "muxBool"(addr := #inSimulate.DO7, i0 := #in7, i1 := false, i2 := true, out => #out7)
   END_RUNG
   // the same network as SCL:
   "muxBool"(addr := #inSimulate.DO7, i0 := #in7, i1 := false, i2 := true, out => #out7);
END_REGION

REGION Network 10
   RUNG wire#powerrail
      "muxBool"(addr := #inSimulate.DO8, i0 := #in8, i1 := false, i2 := true, out => #out8)
   END_RUNG
   // the same network as SCL:
   "muxBool"(addr := #inSimulate.DO8, i0 := #in8, i1 := false, i2 := true, out => #out8);
END_REGION

REGION Network 11
   RUNG wire#powerrail
      "muxBool"(addr := #inSimulate.DO9, i0 := #in9, i1 := false, i2 := true, out => #out9)
   END_RUNG
   // the same network as SCL:
   "muxBool"(addr := #inSimulate.DO9, i0 := #in9, i1 := false, i2 := true, out => #out9);
END_REGION

REGION Network 12
   RUNG wire#powerrail
      "muxBool"(addr := #inSimulate.DO10, i0 := #in10, i1 := false, i2 := true, out => #out10)
   END_RUNG
   // the same network as SCL:
   "muxBool"(addr := #inSimulate.DO10, i0 := #in10, i1 := false, i2 := true, out => #out10);
END_REGION

REGION Network 13
   RUNG wire#powerrail
      "muxBool"(addr := #inSimulate.DO11, i0 := #in11, i1 := false, i2 := true, out => #out11)
   END_RUNG
   // the same network as SCL:
   "muxBool"(addr := #inSimulate.DO11, i0 := #in11, i1 := false, i2 := true, out => #out11);
END_REGION

REGION Network 14
   RUNG wire#powerrail
      "muxBool"(addr := #inSimulate.DO12, i0 := #in12, i1 := false, i2 := true, out => #out12)
   END_RUNG
   // the same network as SCL:
   "muxBool"(addr := #inSimulate.DO12, i0 := #in12, i1 := false, i2 := true, out => #out12);
END_REGION

REGION Network 15
   RUNG wire#powerrail
      "muxBool"(addr := #inSimulate.DO13, i0 := #in13, i1 := false, i2 := true, out => #out13)
   END_RUNG
   // the same network as SCL:
   "muxBool"(addr := #inSimulate.DO13, i0 := #in13, i1 := false, i2 := true, out => #out13);
END_REGION

REGION Network 16
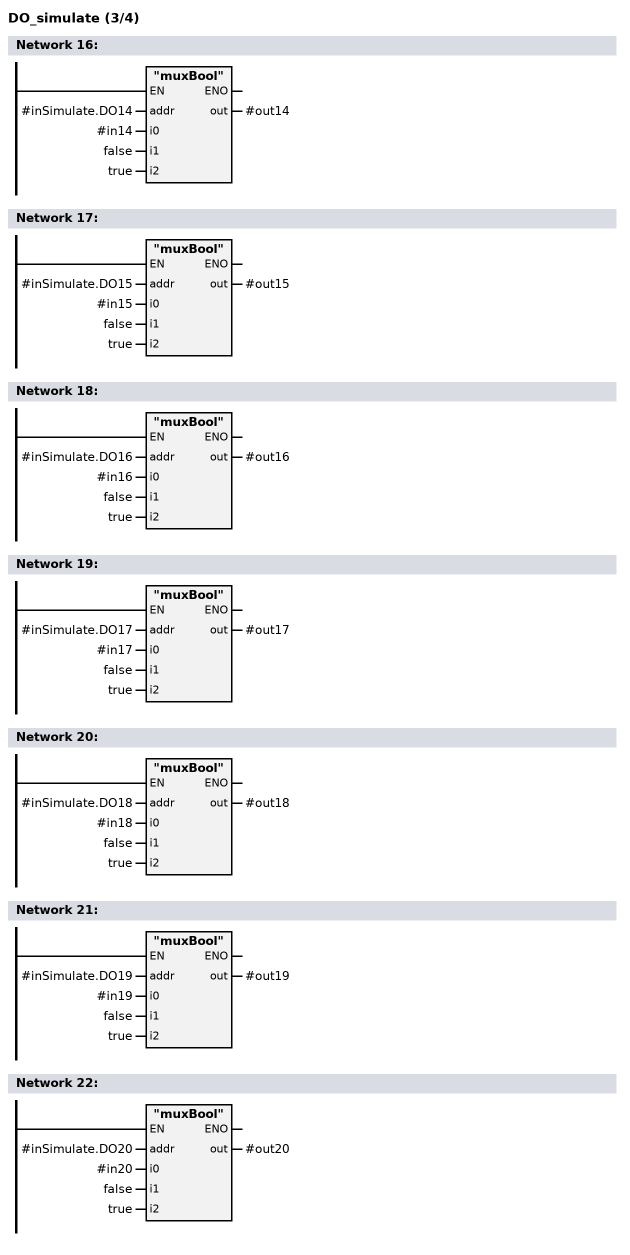
   RUNG wire#powerrail
      "muxBool"(addr := #inSimulate.DO14, i0 := #in14, i1 := false, i2 := true, out => #out14)
   END_RUNG
   // the same network as SCL:
   "muxBool"(addr := #inSimulate.DO14, i0 := #in14, i1 := false, i2 := true, out => #out14);
END_REGION

REGION Network 17
   RUNG wire#powerrail
      "muxBool"(addr := #inSimulate.DO15, i0 := #in15, i1 := false, i2 := true, out => #out15)
   END_RUNG
   // the same network as SCL:
   "muxBool"(addr := #inSimulate.DO15, i0 := #in15, i1 := false, i2 := true, out => #out15);
END_REGION

REGION Network 18
   RUNG wire#powerrail
      "muxBool"(addr := #inSimulate.DO16, i0 := #in16, i1 := false, i2 := true, out => #out16)
   END_RUNG
   // the same network as SCL:
   "muxBool"(addr := #inSimulate.DO16, i0 := #in16, i1 := false, i2 := true, out => #out16);
END_REGION

REGION Network 19
   RUNG wire#powerrail
      "muxBool"(addr := #inSimulate.DO17, i0 := #in17, i1 := false, i2 := true, out => #out17)
   END_RUNG
   // the same network as SCL:
   "muxBool"(addr := #inSimulate.DO17, i0 := #in17, i1 := false, i2 := true, out => #out17);
END_REGION

REGION Network 20
   RUNG wire#powerrail
      "muxBool"(addr := #inSimulate.DO18, i0 := #in18, i1 := false, i2 := true, out => #out18)
   END_RUNG
   // the same network as SCL:
   "muxBool"(addr := #inSimulate.DO18, i0 := #in18, i1 := false, i2 := true, out => #out18);
END_REGION

REGION Network 21
   RUNG wire#powerrail
      "muxBool"(addr := #inSimulate.DO19, i0 := #in19, i1 := false, i2 := true, out => #out19)
   END_RUNG
   // the same network as SCL:
   "muxBool"(addr := #inSimulate.DO19, i0 := #in19, i1 := false, i2 := true, out => #out19);
END_REGION

REGION Network 22
   RUNG wire#powerrail
      "muxBool"(addr := #inSimulate.DO20, i0 := #in20, i1 := false, i2 := true, out => #out20)
   END_RUNG
   // the same network as SCL:
   "muxBool"(addr := #inSimulate.DO20, i0 := #in20, i1 := false, i2 := true, out => #out20);
END_REGION

REGION Network 23
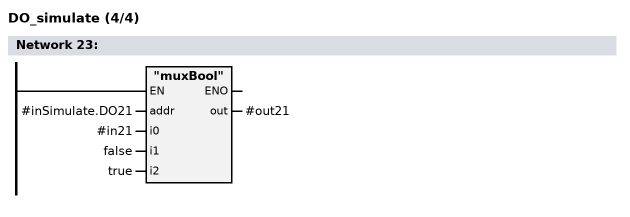
   RUNG wire#powerrail
      "muxBool"(addr := #inSimulate.DO21, i0 := #in21, i1 := false, i2 := true, out => #out21)
   END_RUNG
   // the same network as SCL:
   "muxBool"(addr := #inSimulate.DO21, i0 := #in21, i1 := false, i2 := true, out => #out21);
END_REGION
END_FUNCTION

FUNCTION "muxBool" : Void   // FC3, SCL
{ S7_Optimized_Access := 'TRUE' }
VERSION : 0.1
   VAR_INPUT
      addr : USInt;
      i0 : Bool;
      i1 : Bool;
      i2 : Bool;
   END_VAR
   VAR_OUTPUT
      out : Bool;
   END_VAR
BEGIN
   IF #addr = 1 THEN
       #out := FALSE;
   ELSIF #addr = 2 THEN
       #out := TRUE;
   ELSE
       #out := #i0;
   END_IF;
END_FUNCTION

FUNCTION "AI_simulate" : Void   // FC4, LAD
{ S7_Optimized_Access := 'TRUE' }
VERSION : 0.1
   VAR_INPUT
      in0 : Int;   // upTempLaser1
      in1 : Int;   // upTempLaser2
      in2 : Int;   // upTempCam1
      in3 : Int;   // upTempCam2
      in4 : Int;   // downTempLaser1
      in5 : Int;   // downTempLaser2
      in6 : Int;   // downTempCam1
      in7 : Int;   // downTempCam2
      in8 : Int;   // airTemperatur
      in9 : Int;   // speedRaw
      inOffset : Struct
         upTempLaser1 : Real;   // (Ain0.0)
         upTempLaser2 : Real;   // (Ain0.1)
         upTempCam1 : Real;   // (Ain0.2)
         upTempCam2 : Real;   // (Ain0.3)
         downTempLaser1 : Real;   // (Ain0.4)
         downTempLaser2 : Real;   // (Ain0.5)
         downTempCam1 : Real;   // (Ain0.6)
         downTempCam2 : Real;   // (Ain0.7)
         airTemperatur : Real;   // (Ain1.0)
         speed : Real;   // (Ain2.0)
      END_STRUCT;
      inSimulate : Struct   // Аналоговые входы. 0.0 - симуляция отключена; Либое иное значение включает симуляцию.
         upTempLaser1 : Real;   // (Ain0.0)
         upTempLaser2 : Real;   // (Ain0.1)
         upTempCam1 : Real;   // (Ain0.2)
         upTempCam2 : Real;   // (Ain0.3)
         downTempLaser1 : Real;   // (Ain0.4)
         downTempLaser2 : Real;   // (Ain0.5)
         downTempCam1 : Real;   // (Ain0.6)
         downTempCam2 : Real;   // (Ain0.7)
         airTemperatur : Real;   // (Ain1.0)
         speed : Real;   // (Ain2.0)
      END_STRUCT;
   END_VAR
   VAR_OUTPUT
      out0 : Real;
      out1 : Real;
      out2 : Real;
      out3 : Real;
      out4 : Real;
      out5 : Real;
      out6 : Real;
      out7 : Real;
      out8 : Real;
      out9 : Real;
      out9Min : Bool;
      out9Max : Bool;
   END_VAR
   VAR_TEMP
      b0 : Bool;
      b1 : Bool;
      iAin0 : Real;
      iAin1 : Real;
      iAin2 : Real;
      iAin3 : Real;
      iAin4 : Real;
      iAin5 : Real;
      iAin6 : Real;
      iAin7 : Real;
      iAin8 : Real;
      iAin9 : Real;
      iAin99 : Real;
      err0 : Bool;
      err1 : Bool;
      err00 : Bool;
      err11 : Bool;
      in000 : Bool;
   END_VAR
   VAR_TEMP   // added for the SCL form of the ladder/FBD networks
      _w1 : Bool;
   END_VAR
BEGIN

REGION Network 1 (SCL): Конвертация во флоат, градусы
   #iAin0 := INT_TO_REAL(#in0) / 10;
   #iAin1 := INT_TO_REAL(#in1) / 10;
   #iAin2 := INT_TO_REAL(#in2) / 10;
   #iAin3 := INT_TO_REAL(#in3) / 10;
   #iAin4 := INT_TO_REAL(#in4) / 10;
   #iAin5 := INT_TO_REAL(#in5) / 10;
   #iAin6 := INT_TO_REAL(#in6) / 10;
   #iAin7 := INT_TO_REAL(#in7) / 10;
   #iAin8 := INT_TO_REAL(#in8) / 10;
END_REGION

REGION Network 2 (SCL): Задает смещение
   #out0 := #inOffset.upTempLaser1 + #iAin0;
   #out1 := #inOffset.upTempLaser2 + #iAin1;
   #out2 := #inOffset.upTempCam1 + #iAin2;
   #out3 := #inOffset.upTempCam2 + #iAin3;
   #out4 := #inOffset.downTempLaser1 + #iAin4;
   #out5 := #inOffset.downTempLaser2 + #iAin5;
   #out6 := #inOffset.downTempCam1 + #iAin6;
   #out7 := #inOffset.downTempCam2 + #iAin7;
   #out8 := #inOffset.airTemperatur + #iAin8;
END_REGION

REGION Network 3 (SCL): детектор аварии аналоговых входов

   "READ".warning.overFlowUpLaserAin00 := (#in0 > 2000);
   "READ".warning.underFlowUpLaserAin00 := (#in0 < -500);
   IF "READ".warning.overFlowUpLaserAin00 OR "READ".warning.underFlowUpLaserAin00 THEN
       #out0 := -49.999;
       "Main_PRG".errUpTempLaser1 := TRUE;
   ELSE
       "Main_PRG".errUpTempLaser1 := FALSE;
   END_IF;

   "READ".warning.overFlowUpLaserAin01 := (#in1 > 2000);
   "READ".warning.underFlowUpLaserAin01 := (#in1 < -500);
   IF "READ".warning.overFlowUpLaserAin01 OR "READ".warning.underFlowUpLaserAin01 THEN
       #out1 := -49.999;
       "Main_PRG".errUpTempLaser2 := TRUE;
   ELSE
       "Main_PRG".errUpTempLaser2 := FALSE;
   END_IF;

   "READ".warning.overFlowUpCamAin02 := (#in2 > 2000);
   "READ".warning.underFlowUpCamAin02 := (#in2 < -500);
   IF "READ".warning.overFlowUpCamAin02 OR "READ".warning.underFlowUpCamAin02 THEN
       #out2 := -49.999;
       "Main_PRG".errUpTempCam1 := TRUE;
   ELSE
       "Main_PRG".errUpTempCam1 := FALSE;
   END_IF;

   "READ".warning.overFlowUpCamAin03 := (#in3 > 2000);
   "READ".warning.underFlowUpCamAin03 := (#in3 < -500);
   IF "READ".warning.overFlowUpCamAin03 OR "READ".warning.underFlowUpCamAin03 THEN
       #out3 := -49.999;
       "Main_PRG".errUpTempCam2 := TRUE;
   ELSE
       "Main_PRG".errUpTempCam2 := FALSE;
   END_IF;

   "READ".warning.overFlowDownLaserAin04 := (#in4 > 2000);
   "READ".warning.underFlowDownLaserAin04 := (#in4 < -500);
   IF "READ".warning.overFlowDownLaserAin04 OR "READ".warning.underFlowDownLaserAin04 THEN
       #out4 := -49.999;
       "Main_PRG".errDownTempLaser1 := TRUE;
   ELSE
       "Main_PRG".errDownTempLaser1 := FALSE;
   END_IF;

   "READ".warning.overFlowDownLaserAin05 := (#in5 > 2000);
   "READ".warning.underFlowDownLaserAin05 := (#in5 < -500);
   IF "READ".warning.overFlowDownLaserAin05 OR "READ".warning.underFlowDownLaserAin05 THEN
       #out5 := -49.999;
       "Main_PRG".errDownTempLaser2 := TRUE;
   ELSE
       "Main_PRG".errDownTempLaser2 := FALSE;
   END_IF;

   "READ".warning.overFlowDownCamAin06 := (#in6 > 2000);
   "READ".warning.underFlowDownCamAin06 := (#in6 < -500);
   IF "READ".warning.overFlowDownCamAin06 OR "READ".warning.underFlowDownCamAin06 THEN
       #out6 := -49.999;
       "Main_PRG".errDownTempCam1 := TRUE;
   ELSE
       "Main_PRG".errDownTempCam1 := FALSE;
   END_IF;

   "READ".warning.overFlowDownCamAin07 := (#in7 > 2000);
   "READ".warning.underFlowDownCamAin07 := (#in7 < -500);
   IF "READ".warning.overFlowDownCamAin07 OR "READ".warning.underFlowDownCamAin07 THEN
       #out7 := -49.999;
       "Main_PRG".errDownTempCam2 := TRUE;
   ELSE
       "Main_PRG".errDownTempCam2 := FALSE;
   END_IF;

   "READ".warning.overFlowPneumaticAin10 := (#in8 > 2000);
   "READ".warning.underFlowPneumaticAin10 := (#in8 < -500);
   IF "READ".warning.overFlowPneumaticAin10 OR "READ".warning.underFlowPneumaticAin10 THEN
       #out8 := -49.999;
       "Main_PRG".errAirTemperatur := TRUE;
   ELSE
       "Main_PRG".errAirTemperatur := FALSE;
   END_IF;
END_REGION

REGION Network 4 (SCL): Симуляция (Ain0.0)
   IF #inSimulate.upTempLaser1 <> 0.0 THEN
       #out0 := #inSimulate.upTempLaser1;
       IF (#inSimulate.upTempLaser1 > 0.0) AND (#inSimulate.upTempLaser1 < 0.001) THEN
           #out0 := 0.0;
       END_IF;
   END_IF;
END_REGION

REGION Network 5 (SCL): Симуляция (Ain0.1)
   IF #inSimulate.upTempLaser2 <> 0.0 THEN
       #out1 := #inSimulate.upTempLaser2;
       IF (#inSimulate.upTempLaser2 > 0.0) AND (#inSimulate.upTempLaser2 < 0.001) THEN
           #out1 := 0.0;
       END_IF;
   END_IF;
END_REGION

REGION Network 6 (SCL): Симуляция (Ain0.2)
   IF #inSimulate.upTempCam1 <> 0.0 THEN
       #out2 := #inSimulate.upTempCam1;
       IF (#inSimulate.upTempCam1 > 0.0) AND (#inSimulate.upTempCam1 < 0.001) THEN
           #out2 := 0.0;
       END_IF;
   END_IF;
END_REGION

REGION Network 7 (SCL): Симуляция (Ain0.3)
   IF #inSimulate.upTempCam2 <> 0.0 THEN
       #out3 := #inSimulate.upTempCam2;
       IF (#inSimulate.upTempCam2 > 0.0) AND (#inSimulate.upTempCam2 < 0.001) THEN
           #out3 := 0.0;
       END_IF;
   END_IF;
END_REGION

REGION Network 8 (SCL): Симуляция (Ain0.4)
   IF #inSimulate.downTempLaser1 <> 0.0 THEN
       #out4 := #inSimulate.downTempLaser1;
       IF (#inSimulate.downTempLaser1 > 0.0) AND (#inSimulate.downTempLaser1 < 0.001) THEN
           #out4 := 0.0;
       END_IF;
   END_IF;
END_REGION

REGION Network 9 (SCL): Симуляция (Ain0.5)
   IF #inSimulate.downTempLaser2 <> 0.0 THEN
       #out5 := #inSimulate.downTempLaser2;
       IF (#inSimulate.downTempLaser2 > 0.0) AND (#inSimulate.downTempLaser2 < 0.001) THEN
           #out5 := 0.0;
       END_IF;
   END_IF;
END_REGION

REGION Network 10 (SCL): Симуляция (Ain0.6)
   IF #inSimulate.downTempCam1 <> 0.0 THEN
       #out6 := #inSimulate.downTempCam1;
       IF (#inSimulate.downTempCam1 > 0.0) AND (#inSimulate.downTempCam1 < 0.001) THEN
           #out6 := 0.0;
       END_IF;
   END_IF;
END_REGION

REGION Network 11 (SCL): Симуляция (Ain0.7)
   IF #inSimulate.downTempCam2 <> 0.0 THEN
       #out7 := #inSimulate.downTempCam2;
       IF (#inSimulate.downTempCam2 > 0.0) AND (#inSimulate.downTempCam2 < 0.001) THEN
           #out7 := 0.0;
       END_IF;
   END_IF;
END_REGION

REGION Network 12 (SCL): Симуляция (Ain1.0)
   IF #inSimulate.airTemperatur <> 0.0 THEN
       #out8 := #inSimulate.airTemperatur;
       IF (#inSimulate.airTemperatur > 0.0) AND (#inSimulate.airTemperatur < 0.001) THEN
           #out8 := 0.0;
       END_IF;
   END_IF;
END_REGION

REGION Network 13 (SCL): Симуляция (Ain2.0)
   IF #inSimulate.speed <> 0.0 THEN
       #out9 := #inSimulate.speed;
       #err00 := TRUE;
       IF (#inSimulate.speed > 0.0) AND (#inSimulate.speed < 0.001) THEN
           #out9 := 0.0;
       END_IF;
   END_IF;
END_REGION

REGION Network 14: Пересчет в скорость, метр/мин, для Ain2.0. ADD -- смещение.
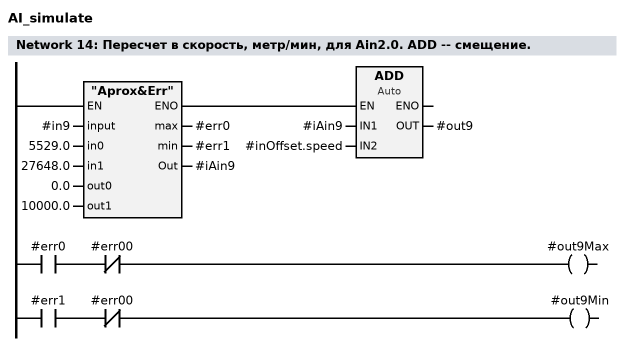
   RUNG wire#powerrail
      "Aprox&Err"(input := #in9, in0 := 5529.0, in1 := 27648.0, out0 := 0.0, out1 := 10000.0, max => #err0, min => #err1, Out => #iAin9)
      Add(in1 := #iAin9, in2 := #inOffset.speed, out => #out9)
   END_RUNG
   RUNG wire#powerrail
      Contact( #err0 )
      I_Contact( #err00 )
      Coil( #out9Max )
   END_RUNG
   RUNG wire#powerrail
      Contact( #err1 )
      I_Contact( #err00 )
      Coil( #out9Min )
   END_RUNG
   // the same network as SCL:
   "Aprox&Err"(input := #in9,
               in0 := 5529.0,
               in1 := 27648.0,
               out0 := 0.0,
               out1 := 10000.0,
               max => #err0,
               min => #err1,
               Out => #iAin9,
               ENO => #_w1);
   IF #_w1 THEN #out9 := #iAin9 + #inOffset.speed; END_IF;
   #out9Max := #err0 AND NOT #err00;
   #out9Min := #err1 AND NOT #err00;
END_REGION
END_FUNCTION

FUNCTION "AO_simulate" : Void   // FC5, LAD
{ S7_Optimized_Access := 'TRUE' }
VERSION : 0.1
   VAR_INPUT
      input : Struct   // Мощность лазеров от 0 до 100%
         writeAll : Real;
         upBlue1 : Real;   // AO0.0
         upBlue2 : Real;   // AO0.1
         upBlue3 : Real;   // AO0.2
         upGreen1 : Real;   // AO0.3
         upGreen2 : Real;   // AO0.4
         upGreen3 : Real;   // AO0.5
         upBlue4 : Real;   // AO0.6
         upBlue5 : Real;   // AO0.7
         upBlue6 : Real;   // AO1.0
         upGreen4 : Real;   // AO1.1
         upGreen5 : Real;   // AO1.2
         upGreen6 : Real;   // AO1.3
         upBlue7 : Real;   // AO1.4
         upBlue8 : Real;   // AO1.5
         upBlue9 : Real;   // AO1.6
         downGreen1 : Real;   // AO2.0
         downGreen2 : Real;   // AO2.1
         downGreen3 : Real;   // AO2.2
         downBlue1 : Real;   // AO2.3
         downBlue2 : Real;   // AO2.4
         downBlue3 : Real;   // AO2.5
         downGreen4 : Real;   // AO2.6
         downGreen5 : Real;   // AO2.7
         downGreen6 : Real;   // AO3.0
         downBlue4 : Real;   // AO3.1
         downBlue5 : Real;   // AO3.2
         downBlue6 : Real;   // AO3.3
         downGreen7 : Real;   // AO3.4
         downGreen8 : Real;   // AO3.5
         downGreen9 : Real;   // AO3.6
      END_STRUCT;
   END_VAR
   VAR_OUTPUT
      out0 : Int;
      out1 : Int;
      out2 : Int;
      out3 : Int;
      out4 : Int;
      out5 : Int;
      out6 : Int;
      out7 : Int;
      out8 : Int;
      out9 : Int;
      out10 : Int;
      out11 : Int;
      out12 : Int;
      out13 : Int;
      out14 : Int;
      out15 : Int;
      out16 : Int;
      out17 : Int;
      out18 : Int;
      out19 : Int;
      out20 : Int;
      out21 : Int;
      out22 : Int;
      out23 : Int;
      out24 : Int;
      out25 : Int;
      out26 : Int;
      out27 : Int;
      out28 : Int;
      out29 : Int;
   END_VAR
   VAR_TEMP
      i : Int;
      in : Array[0..29] of Real;
      apprOut : Array[0..29] of Real;
      out : Array[0..29] of Int;
   END_VAR
BEGIN

REGION Network 1 (SCL): Привязка к массиву
   #in[0] := #input.upBlue1;
   #in[1] := #input.upBlue2;
   #in[2] := #input.upBlue3;
   #in[3] := #input.upGreen1;
   #in[4] := #input.upGreen2;
   #in[5] := #input.upGreen3;
   #in[6] := #input.upBlue4;
   #in[7] := #input.upBlue5;
   #in[8] := #input.upBlue6;
   #in[9] := #input.upGreen4;
   #in[10] := #input.upGreen5;
   #in[11] := #input.upGreen6;
   #in[12] := #input.upBlue7;
   #in[13] := #input.upBlue8;
   #in[14] := #input.upBlue9;
   #in[15] := #input.downGreen1;
   #in[16] := #input.downGreen2;
   #in[17] := #input.downGreen3;
   #in[18] := #input.downBlue1;
   #in[19] := #input.downBlue2;
   #in[20] := #input.downBlue3;
   #in[21] := #input.downGreen4;
   #in[22] := #input.downGreen5;
   #in[23] := #input.downGreen6;
   #in[24] := #input.downBlue4;
   #in[25] := #input.downBlue5;
   #in[26] := #input.downBlue6;
   #in[27] := #input.downGreen7;
   #in[28] := #input.downGreen8;
   #in[29] := #input.downGreen9;
END_REGION

REGION Network 2 (SCL): Конвертирует мощность (%) в код АЦП
   FOR #i := 0 TO 29 DO
       "Approx(real)"(input:=#in[#i],
                      in0:=0.0,
                      in1:=100.0,
                      out0:=0.0,
                      out1:=13824.0,  //13824 == 5Вольт. 27648 == 10Вольт.
                      Out=>#apprOut[#i]); 
       #out[#i] := REAL_TO_INT(#apprOut[#i]);
   END_FOR;
END_REGION

REGION Network 3 (SCL): Извлечение из массива
   #out0 := #out[0];
   #out1 := #out[1];
   #out2 := #out[2];
   #out3 := #out[3];
   #out4 := #out[4];
   #out5 := #out[5];
   #out6 := #out[6];
   #out7 := #out[7];
   #out8 := #out[8];
   #out9 := #out[9];
   #out10 := #out[10];
   #out11 := #out[11];
   #out12 := #out[12];
   #out13 := #out[13];
   #out14 := #out[14];
   #out15 := #out[15];
   #out16 := #out[16];
   #out17 := #out[17];
   #out18 := #out[18];
   #out19 := #out[19];
   #out20 := #out[20];
   #out21 := #out[21];
   #out22 := #out[22];
   #out23 := #out[23];
   #out24 := #out[24];
   #out25 := #out[25];
   #out26 := #out[26];
   #out27 := #out[27];
   #out28 := #out[28];
   #out29 := #out[29];
END_REGION
END_FUNCTION

FUNCTION "Aprox&Err" : Void   // FC6, SCL
{ S7_Optimized_Access := 'TRUE' }
VERSION : 0.1
   VAR_INPUT
      input : Int;
      in0 : Real;
      in1 : Real;
      out0 : Real;
      out1 : Real;
   END_VAR
   VAR_OUTPUT
      max : Bool;
      min : Bool;
      Out : Real;
   END_VAR
   VAR_TEMP
      input_R : Real;
   END_VAR
BEGIN
   #input_R := INT_TO_REAL(#input);
   #Out := (#input_R - #in0) * (#out1 - #out0) / (#in1 - #in0) + #out0;

   IF #input < 4147 THEN
       #min := TRUE;
       #Out := 0;
   END_IF;
   IF #input > 27648 THEN
       #max := TRUE;
       #Out := 10;
   END_IF;
   IF #input < #in0 THEN
       #Out := 0;
   END_IF;
END_FUNCTION

FUNCTION "Approx(real)" : Void   // FC7, SCL
{ S7_Optimized_Access := 'TRUE' }
VERSION : 0.1
   VAR_INPUT
      input : Real;
      in0 : Real;
      in1 : Real;
      out0 : Real;
      out1 : Real;
   END_VAR
   VAR_OUTPUT
      Out : Real;
   END_VAR
BEGIN
   #Out := (#input - #in0) * (#out1 - #out0) / (#in1 - #in0) + #out0;
END_FUNCTION

FUNCTION "error" : Void   // FC8, SCL
{ S7_Optimized_Access := 'TRUE' }
VERSION : 0.1
   VAR_INPUT
      fault : Struct   // 64bit -- Биты аварий
         door1 : Bool;   // Дверь1 -- открыта
         door2 : Bool;   // Дверь2 -- открыта
         power11 : Bool;   // Питание внешних цепей
         power12 : Bool;   // Питание внутренних цепей
         power2 : Bool;   // Питание лазеров, ШВИ, синхробокса, видеокамер
         upLaserTemp : Bool;   // Температура выше аварийного уровня. (Верхний блок лазеров)
         upLaserAllCh : Bool;   // Все каналы измерения температуры неисправны. (Верхний блок лазеров)
         upCamTemp : Bool;   // Температура выше аварийного уровня. (Верхний блок камер)
         upCamAllCh : Bool;   // Все каналы измерения температуры неисправны. (Верхний блок камер)
         downLaserTemp : Bool;   // Температура выше аварийного уровня. (Нижний блок лазеров)
         downLaserAllCh : Bool;   // Все каналы измерения температуры неисправны. (Нижний блок лазеров)
         downCamTemp : Bool;   // Температура выше аварийного уровня. (Нижний блок камер)
         downCamAllCh : Bool;   // Все каналы измерения температуры неисправны. (Нижний блок камер)
         Ain2MinLimit : Bool;   // Вход от велосиметра (4-20мА) ниже уровня 4мА
         Ain2MaxLimit : Bool;   // Вход от велосиметра (4-20мА) выше уровня 20мА
         iniError : Bool;   // Ошибка инициализации.
         reserve0 : Bool;
         reserve1 : Bool;
         reserve2 : Bool;
         reserve3 : Bool;
         reserve4 : Bool;
         reserve5 : Bool;
         reserve6 : Bool;
         reserve7 : Bool;
         reserve8 : Bool;
         reserve9 : Bool;
         reserve10 : Bool;
         reserve11 : Bool;
         reserve12 : Bool;
         reserve13 : Bool;
         reserve14 : Bool;
         reserve15 : Bool;
         reserve16 : Bool;
         reserve17 : Bool;
         reserve18 : Bool;
         reserve19 : Bool;
         reserve20 : Bool;
         reserve21 : Bool;
         reserve22 : Bool;
         reserve23 : Bool;
         reserve24 : Bool;
         reserve25 : Bool;
         reserve26 : Bool;
         reserve27 : Bool;
         reserve28 : Bool;
         reserve29 : Bool;
         reserve30 : Bool;
         reserve31 : Bool;
      END_STRUCT;
   END_VAR
   VAR_OUTPUT
      yes : Bool;
   END_VAR
   VAR_TEMP
      i : USInt;
      "array" : Array[0..63] of Bool;
   END_VAR
BEGIN
   REGION to_Array
       #array[0] := #fault.door1;
       #array[1] := #fault.door2;
       #array[2] := #fault.power11;
       #array[3] := #fault.power12;
       #array[4] := #fault.power2;
       #array[5] := #fault.upLaserTemp;
       #array[6] := #fault.upLaserAllCh;
       #array[7] := #fault.upCamTemp;
       #array[8] := #fault.upCamAllCh;
       #array[9] := #fault.downLaserTemp;
       #array[10] := #fault.downLaserAllCh;
       #array[11] := #fault.downCamTemp;
       #array[12] := #fault.downCamAllCh;
       #array[13] := #fault.Ain2MinLimit;
       #array[14] := #fault.Ain2MaxLimit;
       #array[15] := #fault.iniError;
       #array[16] := #fault.reserve0;
       #array[17] := #fault.reserve1;
       #array[18] := #fault.reserve2;
       #array[19] := #fault.reserve3;
       #array[20] := #fault.reserve4;
       #array[21] := #fault.reserve5;
       #array[22] := #fault.reserve6;
       #array[23] := #fault.reserve7;
       #array[24] := #fault.reserve8;
       #array[25] := #fault.reserve9;
       #array[26] := #fault.reserve10;
       #array[27] := #fault.reserve11;
       #array[28] := #fault.reserve12;
       #array[29] := #fault.reserve13;
       #array[30] := #fault.reserve14;
       #array[31] := #fault.reserve15;
       #array[32] := #fault.reserve16;
       #array[33] := #fault.reserve17;
       #array[34] := #fault.reserve18;
       #array[35] := #fault.reserve19;
       #array[36] := #fault.reserve20;
       #array[37] := #fault.reserve21;
       #array[38] := #fault.reserve22;
       #array[39] := #fault.reserve23;
       #array[40] := #fault.reserve24;
       #array[41] := #fault.reserve25;
       #array[42] := #fault.reserve26;
       #array[43] := #fault.reserve27;
       #array[44] := #fault.reserve28;
       #array[45] := #fault.reserve29;
       #array[46] := #fault.reserve30;
       #array[47] := #fault.reserve31;

   END_REGION ;

   #yes := false;
   FOR #i := 0 TO 63 DO
       IF #array[#i] THEN
           #yes := true;
           EXIT;
       END_IF;
   END_FOR;
END_FUNCTION

FUNCTION "MOD" : Void   // FC9, SCL
{ S7_Optimized_Access := 'TRUE' }
VERSION : 0.1
   VAR_INPUT
      in0 : UDInt;
      in1 : UDInt;
   END_VAR
   VAR_OUTPUT
      Out : USInt;
   END_VAR
BEGIN
   #Out := #in0 - #in1 * (#in0 / #in1);
END_FUNCTION

FUNCTION "warning" : Void   // FC10, SCL
{ S7_Optimized_Access := 'TRUE' }
VERSION : 0.1
   VAR_INPUT
      warnings : Struct
         highTempUpLaser : Bool;   // Температура выше warning уровня. (Верхний блок лазеров)
         highTempUpCam : Bool;   // Температура выше warning уровня. (Верхний блок камер)
         highTempDownLaser : Bool;   // Температура выше warning уровня. (Нижний блок лазеров)
         highTempDownCam : Bool;   // Температура выше warning уровня. (Нижний блок камер)
         highTempPneumatic : Bool;   // Температура выше аварийного уровня. (Воздуха в пневмосистеме)
         power2_1 : Bool;   // Резервированный БП-1 неисправен. (Питание лазеров, ШВИ, синхробокса, видеокамер)
         power2_2 : Bool;   // Резервированный БП-2 неисправен. (Питание лазеров, ШВИ, синхробокса, видеокамер)
         overFlowUpLaserAin00 : Bool;   // Сопротивление датчика 1 температуры выше допустимого (Верхний блок лазеров)
         overFlowUpLaserAin01 : Bool;   // Сопротивление датчика 2 температуры выше допустимого (Верхний блок лазеров)
         overFlowUpCamAin02 : Bool;   // Сопротивление датчика 1 температуры выше допустимого (Верхний блок камер)
         overFlowUpCamAin03 : Bool;   // Сопротивление датчика 2 температуры выше допустимого (Верхний блок камер)
         overFlowDownLaserAin04 : Bool;   // Сопротивление датчика 1 температуры выше допустимого (Нижний блок лазеров)
         overFlowDownLaserAin05 : Bool;   // Сопротивление датчика 2 температуры выше допустимого (Нижний блок лазеров)
         overFlowDownCamAin06 : Bool;   // Сопротивление датчика 1 температуры выше допустимого (Нижний блок камер)
         overFlowDownCamAin07 : Bool;   // Сопротивление датчика 2 температуры выше допустимого (Нижний блок камер)
         overFlowPneumaticAin10 : Bool;   // Сопротивление датчика температуры выше допустимого (Воздух в пневмосистеме)
         underFlowUpLaserAin00 : Bool;   // Сопротивление датчика 1 температуры ниже допустимого (Верхний блок лазеров)
         underFlowUpLaserAin01 : Bool;   // Сопротивление датчика 2 температуры ниже допустимого (Верхний блок лазеров)
         underFlowUpCamAin02 : Bool;   // Сопротивление датчика 1 температуры ниже допустимого (Верхний блок камер)
         underFlowUpCamAin03 : Bool;   // Сопротивление датчика 2 температуры ниже допустимого (Верхний блок камер)
         underFlowDownLaserAin04 : Bool;   // Сопротивление датчика 1 температуры ниже допустимого (Нижний блок лазеров)
         underFlowDownLaserAin05 : Bool;   // Сопротивление датчика 2 температуры ниже допустимого (Нижний блок лазеров)
         underFlowDownCamAin06 : Bool;   // Сопротивление датчика 1 температуры ниже допустимого (Нижний блок камер)
         underFlowDownCamAin07 : Bool;   // Сопротивление датчика 2 температуры ниже допустимого (Нижний блок камер)
         underFlowPneumaticAin10 : Bool;   // Сопротивление датчика температуры ниже допустимого (Воздух в пневмосистеме)
         reserve6 : Bool;
         reserve5 : Bool;
         reserve4 : Bool;
         reserve3 : Bool;
         reserve2 : Bool;
         reserve1 : Bool;
         reserve0 : Bool;
      END_STRUCT;
   END_VAR
   VAR_OUTPUT
      yes : Bool;
   END_VAR
   VAR_TEMP
      i : USInt;
      "array" : Array[0..31] of Bool;
   END_VAR
BEGIN

   REGION warnings
       #array[0] := #warnings.highTempUpLaser;
       #array[1] := #warnings.highTempUpCam;
       #array[2] := #warnings.highTempDownLaser;
       #array[3] := #warnings.highTempDownCam;
       #array[4] := #warnings.highTempPneumatic;
       #array[5] := #warnings.power2_1;
       #array[6] := #warnings.power2_2;
       #array[7] := #warnings.overFlowUpLaserAin00;
       #array[8] := #warnings.overFlowUpLaserAin01;
       #array[9] := #warnings.overFlowUpCamAin02;
       #array[10] := #warnings.overFlowUpCamAin03;
       #array[11] := #warnings.overFlowDownLaserAin04;
       #array[12] := #warnings.overFlowDownLaserAin05;
       #array[13] := #warnings.overFlowDownCamAin06;
       #array[14] := #warnings.overFlowDownCamAin07;
       #array[15] := #warnings.overFlowPneumaticAin10;
       #array[16] := #warnings.underFlowUpLaserAin00;
       #array[17] := #warnings.underFlowUpLaserAin01;
       #array[18] := #warnings.underFlowUpCamAin02;
       #array[19] := #warnings.underFlowUpCamAin03;
       #array[20] := #warnings.underFlowDownLaserAin04;
       #array[21] := #warnings.underFlowDownLaserAin05;
       #array[22] := #warnings.underFlowDownCamAin06;
       #array[23] := #warnings.underFlowDownCamAin07;
       #array[24] := #warnings.underFlowPneumaticAin10;
       #array[25] := #warnings.reserve6;
       #array[26] := #warnings.reserve5;
       #array[27] := #warnings.reserve4;
       #array[28] := #warnings.reserve3;
       #array[29] := #warnings.reserve2;
       #array[30] := #warnings.reserve1;
       #array[31] := #warnings.reserve0;
   END_REGION

   #yes := false;
   FOR #i := 0 TO 31 DO
       IF #array[#i] THEN
           #yes := true;
           EXIT;
       END_IF;
   END_FOR;
END_FUNCTION

FUNCTION "XOR" : Void   // FC11, LAD
{ S7_Optimized_Access := 'TRUE' }
VERSION : 0.1
   VAR_INPUT
      in0 : Bool;
      in1 : Bool;
   END_VAR
   VAR_OUTPUT
      Q : Bool;
   END_VAR
BEGIN

REGION Network 1
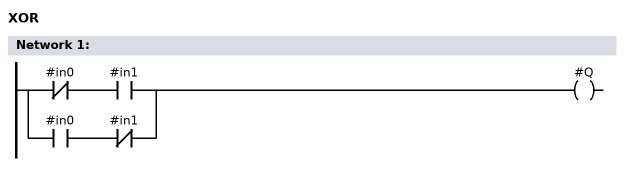
   RUNG wire#powerrail
      I_Contact( #in0 )
      Contact( #in1 )
      wire#w1
      Coil( #Q )
   END_RUNG
   RUNG wire#powerrail
      Contact( #in0 )
      I_Contact( #in1 )
   END_RUNG wire#w1
   // the same network as SCL:
   #Q := (NOT #in0 AND #in1) OR (#in0 AND NOT #in1);
END_REGION
END_FUNCTION

FUNCTION "status" : Void   // FC12, SCL
{ S7_Optimized_Access := 'TRUE' }
VERSION : 0.1
   VAR_INPUT
      "1" : Bool;
      "2" : Bool;
      "3" : Bool;
      "4" : Bool;
      "5" : Bool;
      "6" : Bool;
   END_VAR
   VAR_OUTPUT
      out : Int;
   END_VAR
BEGIN
   #out := 0;

   IF #"1" THEN
       #out := 1;
   END_IF;

   IF #"2" THEN
       #out := 2;
   END_IF;

   IF #"3" THEN
       #out := 3;
   END_IF;

   IF #"4" THEN
       #out := 4;
   END_IF;

   IF #"5" THEN
       #out := 5;
   END_IF;

   IF #"6" THEN
       #out := #out + 10;
   END_IF;
END_FUNCTION

FUNCTION "2OR" : Void   // FC13, LAD
{ S7_Optimized_Access := 'TRUE' }
VERSION : 0.1
   VAR_INPUT
      in0 : Bool;
      in1 : Bool;
   END_VAR
   VAR_OUTPUT
      Q : Bool;
   END_VAR
BEGIN

REGION Network 1
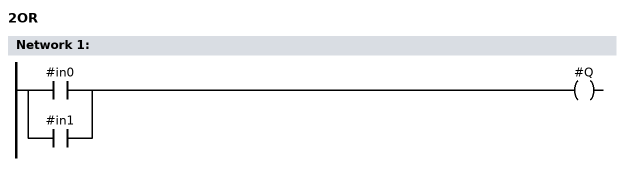
   RUNG wire#powerrail
      Contact( #in0 )
      wire#w1
      Coil( #Q )
   END_RUNG
   RUNG wire#powerrail
      Contact( #in1 )
   END_RUNG wire#w1
   // the same network as SCL:
   #Q := #in0 OR #in1;
END_REGION
END_FUNCTION

FUNCTION "Swap&toInt" : Void   // FC14, LAD
{ S7_Optimized_Access := 'TRUE' }
VERSION : 0.1
   VAR_INPUT
      In : DWord;
   END_VAR
   VAR_OUTPUT
      Out : DInt;
   END_VAR
   VAR_TEMP
      t0 : DWord;
   END_VAR
BEGIN

REGION Network 1
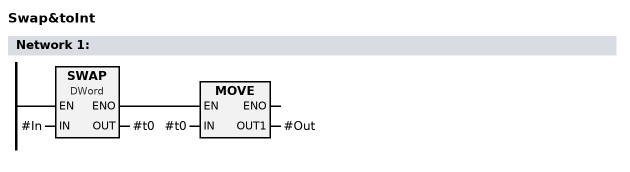
   #t0 := SWAP(#In);
   #Out := #t0;
END_REGION
END_FUNCTION

// folder: Modbus

FUNCTION_BLOCK "Modbus_Client"   // FB15, LAD
{ S7_Optimized_Access := 'TRUE' }
VERSION : 0.1
   VAR_OUTPUT
      error : Bool;
      status : Word;
      noConnect : Bool;
   END_VAR
   VAR
      done : Bool;
      MB_CLIENT_Instance_1 : MB_CLIENT;
      IEC_Timer_0_Instance : TON_TIME;
      IEC_Timer_0_Instance_1 : TON_TIME;
      Blink_Instance : "Blink";
      IEC_Timer_0_Instance_2 : TON_TIME;
      IEC_Timer_0_Instance_3 : TON_TIME;
      IEC_Timer_0_Instance_4 : TON_TIME;
      IEC_Timer_0_Instance_5 : TON_TIME;
      IEC_Timer_0_Instance_6 : TON_TIME;
   END_VAR
   VAR_TEMP
      request : Bool;
      caseH : Bool;
      caseL : Bool;
      laserH : Bool;
      laserL : Bool;
      guageH : Bool;
   END_VAR
BEGIN

REGION Network 1: генератор передачи данных
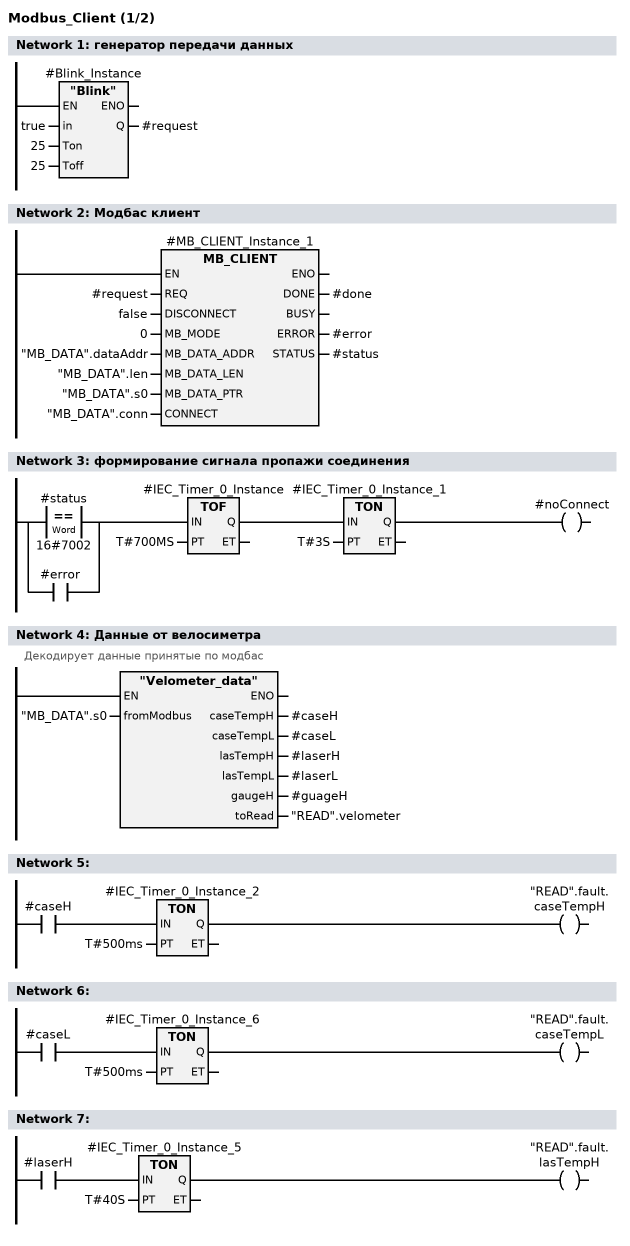
   RUNG wire#powerrail
      #Blink_Instance(in := true, Ton := 25, Toff := 25, Q => #request)
   END_RUNG
   // the same network as SCL:
   #Blink_Instance(in := true, Ton := 25, Toff := 25, Q => #request);   // "Blink"
END_REGION

REGION Network 2: Модбас клиент
   #MB_CLIENT_Instance_1(REQ := #request,   // MB_CLIENT
                         DISCONNECT := false,
                         MB_MODE := 0,
                         MB_DATA_ADDR := "MB_DATA".dataAddr,
                         MB_DATA_LEN := "MB_DATA".len,
                         MB_DATA_PTR := "MB_DATA".s0,
                         CONNECT := "MB_DATA".conn,
                         DONE => #done,
                         ERROR => #error,
                         STATUS => #status);
END_REGION

REGION Network 3: формирование сигнала пропажи соединения
   #IEC_Timer_0_Instance(IN := (#status = 16#7002) OR #error, PT := T#700MS);   // TOF
   #IEC_Timer_0_Instance_1(IN := #IEC_Timer_0_Instance.Q, PT := T#3S);   // TON
   #noConnect := #IEC_Timer_0_Instance_1.Q;
END_REGION

REGION Network 4: Данные от велосиметра
   // Декодирует данные принятые по модбас
   RUNG wire#powerrail
      "Velometer_data"(fromModbus := "MB_DATA".s0, caseTempH => #caseH, caseTempL => #caseL, lasTempH => #laserH, lasTempL => #laserL, gaugeH => #guageH, toRead => "READ".velometer)
   END_RUNG
   // the same network as SCL:
   "Velometer_data"(fromModbus := "MB_DATA".s0,
                    caseTempH => #caseH,
                    caseTempL => #caseL,
                    lasTempH => #laserH,
                    lasTempL => #laserL,
                    gaugeH => #guageH,
                    toRead => "READ".velometer);
END_REGION

REGION Network 5
   #IEC_Timer_0_Instance_2(IN := #caseH, PT := T#500ms);   // TON
   "READ".fault.caseTempH := #IEC_Timer_0_Instance_2.Q;
END_REGION

REGION Network 6
   #IEC_Timer_0_Instance_6(IN := #caseL, PT := T#500ms);   // TON
   "READ".fault.caseTempL := #IEC_Timer_0_Instance_6.Q;
END_REGION

REGION Network 7
   #IEC_Timer_0_Instance_5(IN := #laserH, PT := T#40S);   // TON
   "READ".fault.lasTempH := #IEC_Timer_0_Instance_5.Q;
END_REGION

REGION Network 8
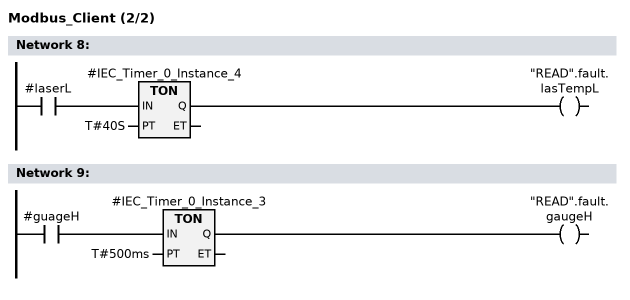
   #IEC_Timer_0_Instance_4(IN := #laserL, PT := T#40S);   // TON
   "READ".fault.lasTempL := #IEC_Timer_0_Instance_4.Q;
END_REGION

REGION Network 9
   #IEC_Timer_0_Instance_3(IN := #guageH, PT := T#500ms);   // TON
   "READ".fault.gaugeH := #IEC_Timer_0_Instance_3.Q;
END_REGION
END_FUNCTION_BLOCK

// folder: Socket_Send

FUNCTION_BLOCK "Sock_RD"   // FB12, LAD
{ S7_Optimized_Access := 'TRUE' }
VERSION : 0.1
   VAR_OUTPUT
      error : Bool;
      status : Word;
   END_VAR
   VAR
      busy : Bool;
      req : Bool;
      IEC_Timer_0_Instance : TON_TIME;
      tt : Int;
   END_VAR
   VAR_TEMP   // added for the SCL form of the ladder/FBD networks
      _w1 : Bool;
   END_VAR
BEGIN

REGION Network 1
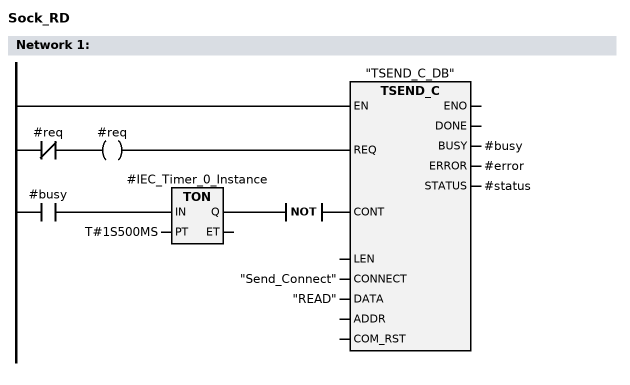
   #_w1 := NOT #req;
   #req := #_w1;
   #IEC_Timer_0_Instance(IN := #busy, PT := T#1S500MS);   // TON
   "TSEND_C_DB"(REQ := #_w1,   // TSEND_C
                CONT := NOT #IEC_Timer_0_Instance.Q,
                CONNECT := "Send_Connect",
                DATA := "READ",
                BUSY => #busy,
                ERROR => #error,
                STATUS => #status);
END_REGION
END_FUNCTION_BLOCK

// folder: Socket_Write

FUNCTION_BLOCK "Sock_WR"   // FB13, LAD
{ S7_Optimized_Access := 'TRUE' }
VERSION : 0.1
   VAR_OUTPUT
      error : Bool;
      stat : Word;
   END_VAR
   VAR
      busyTrcv : Bool;
      fall0 : Bool;
      setLasers_buff : Array[0..9] of Bool;
      DI_buff : Array[0..15] of USInt;
      DO_buff : Array[0..31] of USInt;
      AI_buff : Array[0..9] of Real;
      setTemperatures_buff : Array[0..12] of Real;
      cleanTime_buff : Array[0..1] of Real;
      setPowerLasers_buff : Array[0..30] of Real;
      IEC_Timer_0_Instance_0 : TON_TIME;
      TRCV_C_Instance_0 : TRCV_C;
      IEC_Timer_0_Instance : TON_TIME;
      IEC_Timer_0_Instance_1 : TOF_TIME;
   END_VAR
   VAR_TEMP
      DI_err : Bool;
      DO_err : Bool;
      AI_err : Bool;
      setTemperatures_err : Bool;
      cleanTime_err : Bool;
      setPowerLasers_err : Bool;
      enyValueError : Bool;
      first_start : Bool;
      i0 : USInt;
      i1 : USInt;
      i2 : USInt;
      i3 : USInt;
      i4 : USInt;
      i5 : USInt;
   END_VAR
   VAR_TEMP   // added for the SCL form of the ladder/FBD networks
      _w1 : Bool;
   END_VAR
BEGIN

REGION Network 1
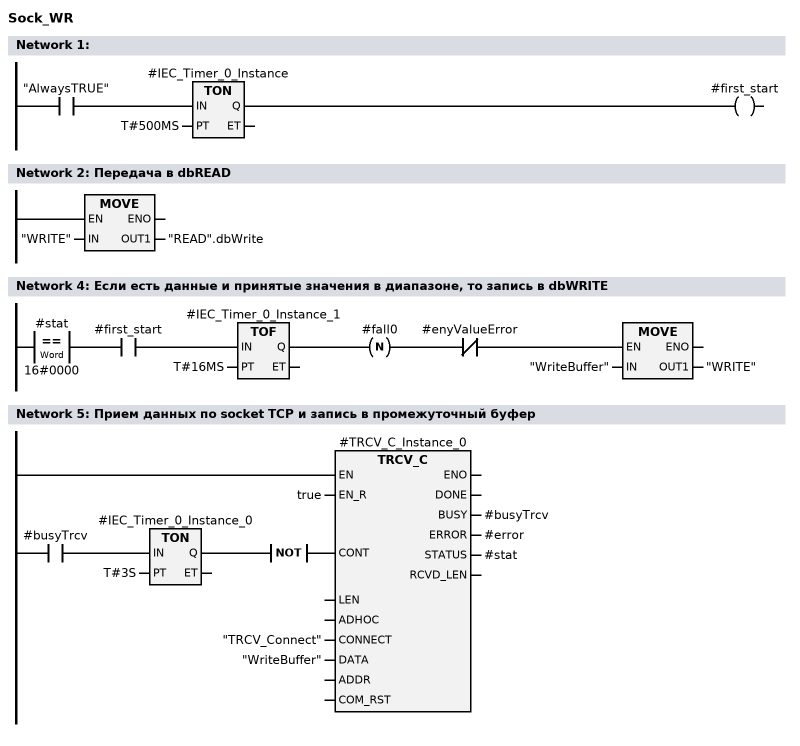
   #IEC_Timer_0_Instance(IN := "AlwaysTRUE", PT := T#500MS);   // TON
   #first_start := #IEC_Timer_0_Instance.Q;
END_REGION

REGION Network 2: Передача в dbREAD
   RUNG wire#powerrail
      Move(in := "WRITE", out1 => "READ".dbWrite)
   END_RUNG
   // the same network as SCL:
   "READ".dbWrite := "WRITE";
END_REGION

REGION Network 3 (SCL): Проверка принятых числел, входят ли они в диапазон

   REGION setLasers
       #setLasers_buff[0] := "WriteBuffer".setLasersManual.upBlueLasers123;
       #setLasers_buff[1] := "WriteBuffer".setLasersManual.upGreenLasers123;
       #setLasers_buff[2] := "WriteBuffer".setLasersManual.upBlueLasers456;
       #setLasers_buff[3] := "WriteBuffer".setLasersManual.upGreenLasers456;
       #setLasers_buff[4] := "WriteBuffer".setLasersManual.upBlueLasers789;
       #setLasers_buff[5] := "WriteBuffer".setLasersManual.downGreenLasers123;
       #setLasers_buff[6] := "WriteBuffer".setLasersManual.downBlueLasers123;
       #setLasers_buff[7] := "WriteBuffer".setLasersManual.downGreenLasers465;
       #setLasers_buff[8] := "WriteBuffer".setLasersManual.downBlueLasers456;
       #setLasers_buff[9] := "WriteBuffer".setLasersManual.downGreenLasers789;
   END_REGION
   REGION DI_buff
       #DI_buff[0] := "WriteBuffer".simulate.DI.DI0;
       #DI_buff[1] := "WriteBuffer".simulate.DI.DI1;
       #DI_buff[2] := "WriteBuffer".simulate.DI.DI2;
       #DI_buff[3] := "WriteBuffer".simulate.DI.DI3;
       #DI_buff[4] := "WriteBuffer".simulate.DI.DI4;
       #DI_buff[5] := "WriteBuffer".simulate.DI.DI5;
       #DI_buff[6] := "WriteBuffer".simulate.DI.DI6;
       #DI_buff[7] := "WriteBuffer".simulate.DI.DI7;
       #DI_buff[8] := "WriteBuffer".simulate.DI.DI8;
       #DI_buff[9] := "WriteBuffer".simulate.DI.DI9;
       #DI_buff[10] := "WriteBuffer".simulate.DI.DI10;
       #DI_buff[11] := "WriteBuffer".simulate.DI.DI11;
       #DI_buff[12] := "WriteBuffer".simulate.DI.DI12;
       #DI_buff[13] := "WriteBuffer".simulate.DI.DI13;
       #DI_buff[14] := "WriteBuffer".simulate.DI.DI14;
       #DI_buff[15] := "WriteBuffer".simulate.DI.DI15;
   END_REGION
   REGION DO_buff
       #DO_buff[0] := "WriteBuffer".simulate."DO".DO0;
       #DO_buff[1] := "WriteBuffer".simulate."DO".DO1;
       #DO_buff[2] := "WriteBuffer".simulate."DO".DO2;
       #DO_buff[3] := "WriteBuffer".simulate."DO".DO3;
       #DO_buff[4] := "WriteBuffer".simulate."DO".DO4;
       #DO_buff[5] := "WriteBuffer".simulate."DO".DO5;
       #DO_buff[6] := "WriteBuffer".simulate."DO".DO6;
       #DO_buff[7] := "WriteBuffer".simulate."DO".DO7;
       #DO_buff[8] := "WriteBuffer".simulate."DO".DO8;
       #DO_buff[9] := "WriteBuffer".simulate."DO".DO9;
       #DO_buff[10] := "WriteBuffer".simulate."DO".DO10;
       #DO_buff[11] := "WriteBuffer".simulate."DO".DO11;
       #DO_buff[12] := "WriteBuffer".simulate."DO".DO12;
       #DO_buff[13] := "WriteBuffer".simulate."DO".DO13;
       #DO_buff[14] := "WriteBuffer".simulate."DO".DO14;
       #DO_buff[15] := "WriteBuffer".simulate."DO".DO15;
       #DO_buff[16] := "WriteBuffer".simulate."DO".DO16;
       #DO_buff[17] := "WriteBuffer".simulate."DO".DO17;
       #DO_buff[18] := "WriteBuffer".simulate."DO".DO18;
       #DO_buff[19] := "WriteBuffer".simulate."DO".DO19;
       #DO_buff[20] := "WriteBuffer".simulate."DO".DO20;
       #DO_buff[21] := "WriteBuffer".simulate."DO".DO21;
       #DO_buff[22] := "WriteBuffer".simulate."DO".DO22;
       #DO_buff[23] := "WriteBuffer".simulate."DO".DO23;
       #DO_buff[24] := "WriteBuffer".simulate."DO".DO24;
       #DO_buff[25] := "WriteBuffer".simulate."DO".DO25;
       #DO_buff[26] := "WriteBuffer".simulate."DO".DO26;
       #DO_buff[27] := "WriteBuffer".simulate."DO".DO27;
       #DO_buff[28] := "WriteBuffer".simulate."DO".DO28;
       #DO_buff[29] := "WriteBuffer".simulate."DO".DO29;
       #DO_buff[30] := "WriteBuffer".simulate."DO".DO30;
       #DO_buff[31] := "WriteBuffer".simulate."DO".DO31;
   END_REGION
   REGION AI_buff
       #AI_buff[0] := "WriteBuffer".simulate.AI.upTempLaser1;
       #AI_buff[1] := "WriteBuffer".simulate.AI.upTempLaser2;
       #AI_buff[2] := "WriteBuffer".simulate.AI.upTempCam1;
       #AI_buff[3] := "WriteBuffer".simulate.AI.upTempCam2;
       #AI_buff[4] := "WriteBuffer".simulate.AI.downTempLaser1;
       #AI_buff[5] := "WriteBuffer".simulate.AI.downTempLaser2;
       #AI_buff[6] := "WriteBuffer".simulate.AI.downTempCam1;
       #AI_buff[7] := "WriteBuffer".simulate.AI.downTempCam2;
       #AI_buff[8] := "WriteBuffer".simulate.AI.airTemperatur;
       #AI_buff[9] := "WriteBuffer".simulate.AI.reserv;
   END_REGION
   REGION setTemperatures_buff
       #setTemperatures_buff[0] := "WriteBuffer".setTemperatures.faultUpLaser;
       #setTemperatures_buff[1] := "WriteBuffer".setTemperatures.faultUpCam;
       #setTemperatures_buff[2] := "WriteBuffer".setTemperatures.faultDownLaser;
       #setTemperatures_buff[3] := "WriteBuffer".setTemperatures.faultDownCam;
       #setTemperatures_buff[4] := "WriteBuffer".setTemperatures.warnAir;
       #setTemperatures_buff[5] := "WriteBuffer".setTemperatures.warnUpLaser;
       #setTemperatures_buff[6] := "WriteBuffer".setTemperatures.warnUpCam;
       #setTemperatures_buff[7] := "WriteBuffer".setTemperatures.warnDownLaser;
       #setTemperatures_buff[8] := "WriteBuffer".setTemperatures.warnDownCam;
       #setTemperatures_buff[9] := "WriteBuffer".setTemperatures.reserv0;
   END_REGION
   REGION cleanTime_buff
       #cleanTime_buff[0] := "WriteBuffer".cleanTime.tOnS;
       #cleanTime_buff[1] := "WriteBuffer".cleanTime.tOffMin;
   END_REGION
   REGION setPowerLasers_buff
       #setPowerLasers_buff[0] := "WriteBuffer".setPowerLasers.writeAll;
       #setPowerLasers_buff[1] := "WriteBuffer".setPowerLasers.upBlue1;
       #setPowerLasers_buff[2] := "WriteBuffer".setPowerLasers.upBlue2;
       #setPowerLasers_buff[3] := "WriteBuffer".setPowerLasers.upBlue3;
       #setPowerLasers_buff[4] := "WriteBuffer".setPowerLasers.upGreen1;
       #setPowerLasers_buff[5] := "WriteBuffer".setPowerLasers.upGreen2;
       #setPowerLasers_buff[6] := "WriteBuffer".setPowerLasers.upGreen3;
       #setPowerLasers_buff[7] := "WriteBuffer".setPowerLasers.upBlue4;
       #setPowerLasers_buff[8] := "WriteBuffer".setPowerLasers.upBlue5;
       #setPowerLasers_buff[9] := "WriteBuffer".setPowerLasers.upBlue6;
       #setPowerLasers_buff[10] := "WriteBuffer".setPowerLasers.upGreen4;
       #setPowerLasers_buff[11] := "WriteBuffer".setPowerLasers.upGreen5;
       #setPowerLasers_buff[12] := "WriteBuffer".setPowerLasers.upGreen6;
       #setPowerLasers_buff[13] := "WriteBuffer".setPowerLasers.upBlue7;
       #setPowerLasers_buff[14] := "WriteBuffer".setPowerLasers.upBlue8;
       #setPowerLasers_buff[15] := "WriteBuffer".setPowerLasers.upBlue9;
       #setPowerLasers_buff[16] := "WriteBuffer".setPowerLasers.downGreen1;
       #setPowerLasers_buff[17] := "WriteBuffer".setPowerLasers.downGreen2;
       #setPowerLasers_buff[18] := "WriteBuffer".setPowerLasers.downGreen3;
       #setPowerLasers_buff[19] := "WriteBuffer".setPowerLasers.downBlue1;
       #setPowerLasers_buff[20] := "WriteBuffer".setPowerLasers.downBlue2;
       #setPowerLasers_buff[21] := "WriteBuffer".setPowerLasers.downBlue3;
       #setPowerLasers_buff[22] := "WriteBuffer".setPowerLasers.downGreen4;
       #setPowerLasers_buff[23] := "WriteBuffer".setPowerLasers.downGreen5;
       #setPowerLasers_buff[24] := "WriteBuffer".setPowerLasers.downGreen6;
       #setPowerLasers_buff[25] := "WriteBuffer".setPowerLasers.downBlue4;
       #setPowerLasers_buff[26] := "WriteBuffer".setPowerLasers.downBlue5;
       #setPowerLasers_buff[27] := "WriteBuffer".setPowerLasers.downBlue6;
       #setPowerLasers_buff[28] := "WriteBuffer".setPowerLasers.downGreen7;
       #setPowerLasers_buff[29] := "WriteBuffer".setPowerLasers.downGreen8;
       #setPowerLasers_buff[30] := "WriteBuffer".setPowerLasers.downGreen9;
   END_REGION

   FOR #i0 := 0 TO 15 DO
       IF #DI_buff[#i0] > 2 THEN
           #DI_err := true;
           EXIT;
       END_IF;
   END_FOR;

   FOR #i1 := 0 TO 31 DO
       IF #DO_buff[#i1] > 2 THEN
           #DO_err := true;
           EXIT;
       END_IF;
   END_FOR;

   FOR #i2 := 0 TO 9 DO
       IF (#AI_buff[#i2] < -30.0) OR (#AI_buff[#i2] > 150) THEN
           #AI_err := true;
           EXIT;
       END_IF;
   END_FOR;

   FOR #i3 := 0 TO 9 DO
       IF (#setTemperatures_buff[#i3] < -30.0) OR (#setTemperatures_buff[#i3] > 150) THEN
           #setTemperatures_err := true;
           EXIT;
       END_IF;
   END_FOR;

   FOR #i4 := 0 TO 1 DO
       IF (#cleanTime_buff[#i4] < 0) OR (#cleanTime_buff[#i4] > 10000) THEN
           #cleanTime_err := true;
           EXIT;
       END_IF;
   END_FOR;

   FOR #i5 := 0 TO 30 DO
       IF (#setPowerLasers_buff[#i5] < 0) OR (#setPowerLasers_buff[#i5] > 100) THEN
           #setPowerLasers_err := true;
           EXIT;
       END_IF;
   END_FOR;

   #enyValueError := #DI_err OR #DO_err OR #AI_err OR #setTemperatures_err OR #cleanTime_err OR #setPowerLasers_err;
END_REGION

REGION Network 4: Если есть данные и принятые значения в диапазоне, то запись в dbWRITE
   #IEC_Timer_0_Instance_1(IN := (#stat = 16#0000) AND #first_start, PT := T#16MS);   // TOF
   #_w1 := NOT #IEC_Timer_0_Instance_1.Q AND #fall0;   // falling edge
   #fall0 := #IEC_Timer_0_Instance_1.Q;
   IF #_w1 AND NOT #enyValueError THEN "WRITE" := "WriteBuffer"; END_IF;
END_REGION

REGION Network 5: Прием данных по socket TCP и запись в промежуточный буфер
   #IEC_Timer_0_Instance_0(IN := #busyTrcv, PT := T#3S);   // TON
   #TRCV_C_Instance_0(EN_R := true,   // TRCV_C
                      CONT := NOT #IEC_Timer_0_Instance_0.Q,
                      CONNECT := "TRCV_Connect",
                      DATA := "WriteBuffer",
                      BUSY => #busyTrcv,
                      ERROR => #error,
                      STATUS => #stat);
END_REGION
END_FUNCTION_BLOCK

// folder: Velosimeter

FUNCTION "Velometer_data" : Void   // FC15, LAD
{ S7_Optimized_Access := 'TRUE' }
VERSION : 0.1
   VAR_INPUT
      fromModbus : Struct
         dw0 : Struct
            b0 : Bool;
            b1 : Bool;
            b2 : Bool;
            b3 : Bool;
            b4 : Bool;
            b5 : Bool;
            b6 : Bool;
            b7 : Bool;
            b8 : Bool;
            b9 : Bool;
            b10 : Bool;
            b11 : Bool;
            b12 : Bool;
            b13 : Bool;
            b14 : Bool;
            b15 : Bool;
         END_STRUCT;
         dw1 : Struct
            b0 : Bool;
            b1 : Bool;
            b2 : Bool;
            b3 : Bool;
            b4 : Bool;
            b5 : Bool;
            b6 : Bool;
            b7 : Bool;
            b8 : Bool;
            b9 : Bool;
            b10 : Bool;
            b11 : Bool;
            b12 : Bool;
            b13 : Bool;
            b14 : Bool;
            b15 : Bool;
         END_STRUCT;
         "dw2&3" : DWord;
         "dw4&5" : DWord;
         "dw6&7" : DWord;
         "dw8&9" : DWord;
         "dw10&11" : DWord;
         "dw12&13" : DWord;
         dw14 : Word;
         dw15 : Word;
         dw16 : Word;
         dw17 : Word;
      END_STRUCT;
   END_VAR
   VAR_OUTPUT
      caseTempH : Bool;
      caseTempL : Bool;
      lasTempH : Bool;
      lasTempL : Bool;
      gaugeH : Bool;
      toRead : Struct
         dw0 : Struct
            measMode : Bool;   // Measurement mode. 0=Normal;1=Batch
            resolut : Bool;   // Resolution of length output. 0=length 0.0001;1=length 0.1
            speedResp : Bool;   // Speed reponse for pulse and analogue output. 0=Instant;1=Averaged
            b3 : Bool;
            b4 : Bool;
            b5 : Bool;
            b6 : Bool;
            b7 : Bool;
            measLen1 : Bool;   // 1=>Preset
            measLen2 : Bool;   // 1=>Preset
            b10 : Bool;
            laserOn : Bool;   // 1= ON;0=OFF
            readingSpeed : Bool;   // 1=Valid;0=Invalid
            objectDetect : Bool;   // 1=Object detected;0=No object
            reading : Bool;   // Good reading status. 1=Lower than threshold;0=OK
            b15 : Bool;
         END_STRUCT;
         dw1 : Struct
            gaugeOk : Bool;   // 1=OK;0=Failed
            lasTempH : Bool;   // Laser temperature too high. 1=Too high;0=OK
            lasTempL : Bool;   // Laser temperature too low. 1=Too low;0=OK
            caseTempH : Bool;   // Case temperature too high. 1=Too low;0=OK
            caseTempL : Bool;   // Case temperature too low. 1=Too low;0=OK
            reflectionH : Bool;   // Light reflection too strong. 1=Too low;0=OK
            gaugeH : Bool;   // Gauge too hot. 1=Too low;0=OK
            b7 : Bool;
            b8 : Bool;
            b9 : Bool;
            b10 : Bool;
            b11 : Bool;
            b12 : Bool;
            b13 : Bool;
            b14 : Bool;
            b15 : Bool;
         END_STRUCT;
         averSpeed : Real;   // Отфильтрованная скорость
         instSpeed : Real;   // Мгновенная скорость
         totalLen : Real;   // Общая длина
         batchLen : Real;   // длина партии
         lastLen : Real;   // предыдущая сохраненная длина
         reelNum : DInt;   // номер измерения
         batchNum : Int;   // 0~65535
         readingLavel : Int;   // 0~100%. Качество фокуса и отраженного сигнала
         SNR : Int;   // 0~65535
         SLX : Int;   // ±200mm
      END_STRUCT;
   END_VAR
   VAR_TEMP
      t0 : DInt;
      t1 : DInt;
      t2 : DInt;
      t3 : DInt;
      t4 : DInt;
      t5 : DInt;
      t6 : DInt;
   END_VAR
BEGIN

REGION Network 1
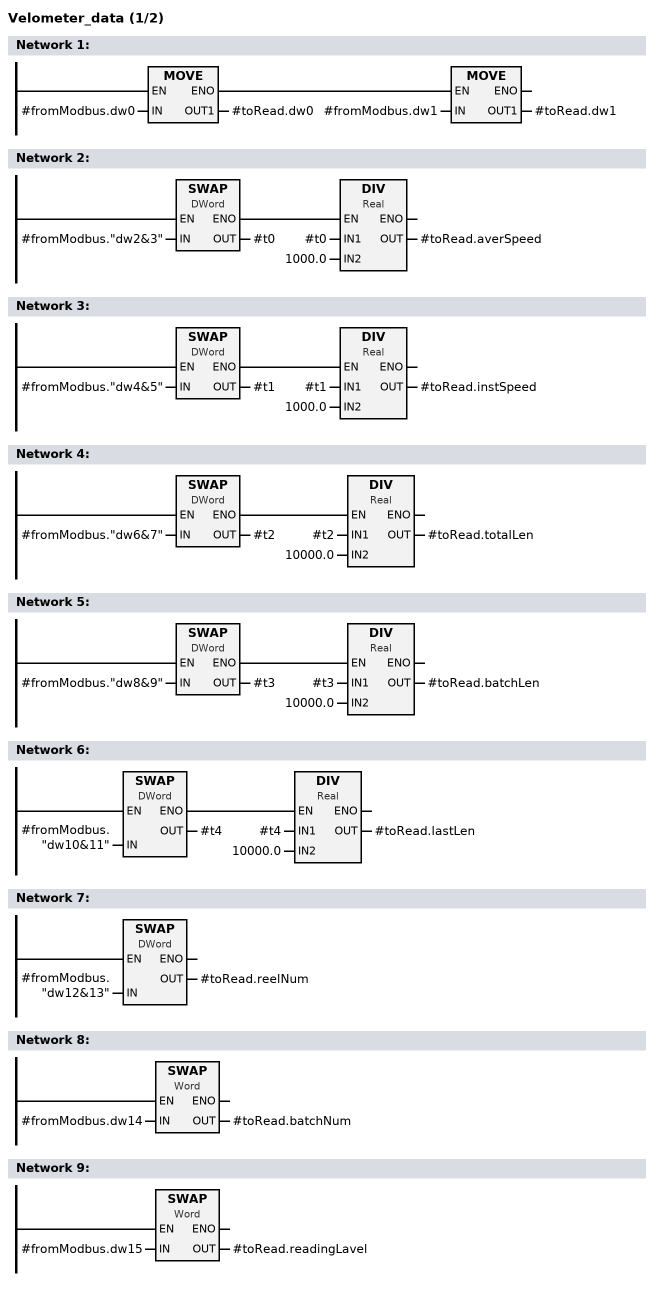
   RUNG wire#powerrail
      { S7_GenerateENO := "TRUE" } Move(in := #fromModbus.dw0, out1 => #toRead.dw0)
      { S7_GenerateENO := "TRUE" } Move(in := #fromModbus.dw1, out1 => #toRead.dw1)
   END_RUNG
   // the same network as SCL:
   // ENO of a box is taken as its EN; it also drops when the box reports an error
   #toRead.dw0 := #fromModbus.dw0;
   #toRead.dw1 := #fromModbus.dw1;
END_REGION

REGION Network 2
   #t0 := SWAP(#fromModbus."dw2&3");
   #toRead.averSpeed := #t0 / 1000.0;
END_REGION

REGION Network 3
   #t1 := SWAP(#fromModbus."dw4&5");
   #toRead.instSpeed := #t1 / 1000.0;
END_REGION

REGION Network 4
   #t2 := SWAP(#fromModbus."dw6&7");
   #toRead.totalLen := #t2 / 10000.0;
END_REGION

REGION Network 5
   #t3 := SWAP(#fromModbus."dw8&9");
   #toRead.batchLen := #t3 / 10000.0;
END_REGION

REGION Network 6
   #t4 := SWAP(#fromModbus."dw10&11");
   #toRead.lastLen := #t4 / 10000.0;
END_REGION

REGION Network 7
   #toRead.reelNum := SWAP(#fromModbus."dw12&13");
END_REGION

REGION Network 8
   #toRead.batchNum := SWAP(#fromModbus.dw14);
END_REGION

REGION Network 9
   #toRead.readingLavel := SWAP(#fromModbus.dw15);
END_REGION

REGION Network 10
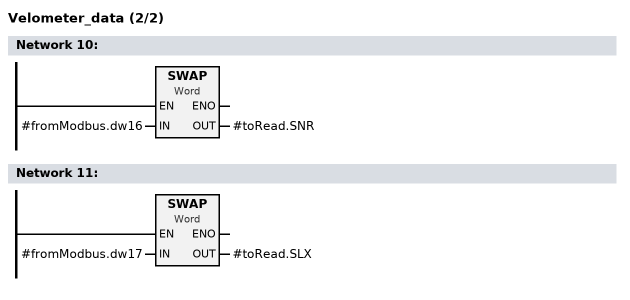
   #toRead.SNR := SWAP(#fromModbus.dw16);
END_REGION

REGION Network 11
   #toRead.SLX := SWAP(#fromModbus.dw17);
END_REGION

REGION Network 12 (SCL)
   #caseTempH := #toRead.dw1.caseTempH;
   #caseTempL := #toRead.dw1.caseTempL;
   #lasTempH := #toRead.dw1.lasTempH;
   #lasTempL := #toRead.dw1.lasTempL;
   #gaugeH := #toRead.dw1.gaugeH;
END_REGION
END_FUNCTION